	IF NOT (WB_PUD.SF_Close AND WB_PUD.State = 0) THEN WB_PUD.B_Close := TRUE; Init := FALSE; END_IF
	IF NOT (WB_PAF.SF_Close AND WB_PAF.State = 0) THEN WB_PAF.B_Close := TRUE; Init := FALSE; END_IF
	IF NOT (WB_SUD.SF_Close AND WB_SUD.State = 0) THEN WB_SUD.B_Close := TRUE; Init := FALSE; END_IF
	IF NOT (WB_SAF.SF_Close AND WB_SAF.State = 0) THEN WB_SAF.B_Close := TRUE; Init := FALSE; END_IF

	WB_A.B_Close := FALSE;
	WB_B.B_Close := FALSE;
	WB_C.B_Close := FALSE;
	WB_D.B_Close := FALSE;
	WB_E.B_Close := FALSE;
	WB_F.B_Close := FALSE;
	WB_G.B_Close := FALSE;
	WB_H.B_Close := FALSE;
	WB_I.B_Close := FALSE;
	WB_J.B_Close := FALSE;
	WB_K.B_Close := FALSE;
	WB_L.B_Close := FALSE;
	WB_M.B_Close := FALSE;
	WB_N.B_Close := FALSE;
	WB_R.B_Close := FALSE;
	WB_S.B_Close := FALSE;

	WB_PUD.B_Close := FALSE;
	WB_PAF.B_Close := FALSE;
	WB_SUD.B_Close := FALSE;
	WB_SAF.B_Close := FALSE;

	IF NOT (WB_A.SF_Open AND WB_A.State = 0) THEN WB_A.B_Open := TRUE; Init := FALSE; END_IF
	IF NOT (WB_B.SF_Open AND WB_B.State = 0) THEN WB_B.B_Open := TRUE; Init := FALSE; END_IF
	IF NOT (WB_C.SF_Open AND WB_C.State = 0) THEN WB_C.B_Open := TRUE; Init := FALSE; END_IF
	IF NOT (WB_D.SF_Open AND WB_D.State = 0) THEN WB_D.B_Open := TRUE; Init := FALSE; END_IF
	IF NOT (WB_E.SF_Open AND WB_E.State = 0) THEN WB_E.B_Open := TRUE; Init := FALSE; END_IF
	IF NOT (WB_F.SF_Open AND WB_F.State = 0) THEN WB_F.B_Open := TRUE; Init := FALSE; END_IF
	IF NOT (WB_G.SF_Open AND WB_G.State = 0) THEN WB_G.B_Open := TRUE; Init := FALSE; END_IF
	IF NOT (WB_H.SF_Open AND WB_H.State = 0) THEN WB_H.B_Open := TRUE; Init := FALSE; END_IF
	IF NOT (WB_I.SF_Open AND WB_I.State = 0) THEN WB_I.B_Open := TRUE; Init := FALSE; END_IF
	IF NOT (WB_J.SF_Open AND WB_J.State = 0) THEN WB_J.B_Open := TRUE; Init := FALSE; END_IF
	IF NOT (WB_K.SF_Open AND WB_K.State = 0) THEN WB_K.B_Open := TRUE; Init := FALSE; END_IF
	IF NOT (WB_L.SF_Open AND WB_L.State = 0) THEN WB_L.B_Open := TRUE; Init := FALSE; END_IF
	IF NOT (WB_M.SF_Open AND WB_M.State = 0) THEN WB_M.B_Open := TRUE; Init := FALSE; END_IF
	IF NOT (WB_N.SF_Open AND WB_N.State = 0) THEN WB_N.B_Open := TRUE; Init := FALSE; END_IF
	IF NOT (WB_R.SF_Open AND WB_R.State = 0) THEN WB_R.B_Open := TRUE; Init := FALSE; END_IF
	IF NOT (WB_S.SF_Open AND WB_S.State = 0) THEN WB_S.B_Open := TRUE; Init := FALSE; END_IF

	IF NOT (WB_PUD.SF_Open AND WB_PUD.State = 0) THEN WB_PUD.B_Open := TRUE; Init := FALSE; END_IF
	IF NOT (WB_PAF.SF_Open AND WB_PAF.State = 0) THEN WB_PAF.B_Open := TRUE; Init := FALSE; END_IF
	IF NOT (WB_SUD.SF_Open AND WB_SUD.State = 0) THEN WB_SUD.B_Open := TRUE; Init := FALSE; END_IF
	IF NOT (WB_SAF.SF_Open AND WB_SAF.State = 0) THEN WB_SAF.B_Open := TRUE; Init := FALSE; END_IF

*)
END_FUNCTION_BLOCK

(* POU FB/FB_WB_VALVE, ST *)
FUNCTION_BLOCK FB_WB_VALVE
VAR_INPUT
	Enable : BOOL;
	Manual : BOOL;

	B_Open  : BOOL;
	B_Close : BOOL;
	SF_Open  : BOOL;
	SF_Close : BOOL;

END_VAR
VAR_IN_OUT
	P   : ST_SENSOR_BAR;
	CFG : ST_WB_VALVE_CFG;
END_VAR
VAR_OUTPUT
	OUT_Open  : BOOL;
	OUT_Close : BOOL;

	OUT_HP    : BYTE;
END_VAR
VAR
	State : WORD;

	IN_Hmi_Open  : BOOL;
	IN_Hmi_Close : BOOL;

	SI_Open  : FB_SMART_INPUT;
	SI_Close : FB_SMART_INPUT;

	SI_Hmi_Open  : FB_SMART_INPUT;
	SI_Hmi_Close : FB_SMART_INPUT;

	TimeCnt : REAL;
	TimeOut : BOOL;

END_VAR
(*Check Inputs*)
SI_Open (In:= B_Open , T_Cont:= T#0ms, T_DClk:= T#0ms);
SI_Close(In:= B_Close, T_Cont:= T#0ms, T_DClk:= T#0ms);

SI_Hmi_Open (In:= IN_Hmi_Open , T_Cont:= T#0ms, T_DClk:= T#0ms);
SI_Hmi_Close(In:= IN_Hmi_Close, T_Cont:= T#0ms, T_DClk:= T#0ms);

IF NOT Enable THEN
	OUT_Open  := FALSE;
	OUT_Close := FALSE;
	OUT_HP    := 0;

	TimeCnt := 0.0;
	State   := 0;
	RETURN;
END_IF

(*Check Time*)
TimeOut := TimeOut OR ( CFG.TimeMax > 0  AND TimeCnt > CFG.TimeMax );
TimeCnt := TimeCnt + CFG.Cycle;

(*Working States*)
CASE State OF

(*Init State*)
0:
	OUT_Open  := FALSE;
	OUT_Close := FALSE;
	OUT_HP    := 0;

	(*Manual*)
	IF Manual THEN
		IF SI_Hmi_Open.Event = INIT_CONTINUOUS AND NOT P.AlMax THEN
			OUT_Open  := TRUE;
			OUT_HP    := 1;
	
			TimeOut := FALSE; (*Reset TimeOut Error*)
			State   := 1001;  (*Next State*)

		ELSIF SI_Hmi_Close.Event = INIT_CONTINUOUS AND NOT P.AlMax THEN
			OUT_Close := TRUE;
			OUT_HP    := 1;

			TimeOut := FALSE; (*Reset TimeOut Error*)
			State   := 1002;  (*Next State*)

		END_IF

	(*Automatico*)
	ELSE
		IF SI_Open.Event = INIT_CONTINUOUS AND NOT P.AlMax THEN
			OUT_Open  := TRUE;
			OUT_HP    := CFG.HP;

			TimeOut := FALSE; (*Reset TimeOut Error*)
			State   := 1010;  (*Next State*)

		ELSIF SI_Close.Event = INIT_CONTINUOUS AND NOT P.AlMax THEN
			OUT_Close := TRUE;
			OUT_HP    := CFG.HP;

			TimeOut := FALSE; (*Reset TimeOut Error*)
			State   := 1020;  (*Next State*)

		END_IF
	END_IF

    TimeCnt := 0.0; (*Time Count*)

(*Manual OPEN*)
1001:
	(*End*)
	IF SI_Hmi_Open.Event <> NONE OR SI_Hmi_Close.Event <> NONE OR TimeOut OR NOT Manual OR P.AlMax THEN
		OUT_Open  := FALSE;
		OUT_HP    := 0;
		State     := 0; (*Next State*)

	END_IF

(*Manual CLOSE*)
1002:
	(*End*)
	IF SI_Hmi_Open.Event <> NONE OR SI_Hmi_Close.Event <> NONE OR TimeOut OR NOT Manual OR P.AlMax THEN
		OUT_Close := FALSE;
		OUT_HP    := 0;
		State     := 0; (*Next State*)

	END_IF

(*Auto OPEN*)
1010:
	(*End*)
	IF SI_Open.Event <> NONE OR TimeOut OR Manual OR P.AlMax THEN
		OUT_Open  := FALSE;
		OUT_HP    := 0;
		State     := 0; (*Next State*)

	ELSIF SI_Close.Event = INIT_CONTINUOUS THEN
		OUT_Open  := FALSE;
		OUT_Close := TRUE;
		State     := 1020; (*Next State*)

	ELSIF SF_Open THEN
		TimeCnt   := 0.0;
		State     := 1011; (*Next State*)

	END_IF

(*Push OPEN*)
1011:
	(*End*)
	IF SI_Open.Event <> NONE OR TimeOut OR TimeCnt > CFG.PushTime OR (CFG.PushP > 0 AND P.Bar > CFG.PushP) OR Manual OR P.AlMax THEN
		OUT_Open  := FALSE;
		OUT_HP    := 0;
		State     := 0; (*Next State*)

	ELSIF SI_Close.Event = INIT_CONTINUOUS THEN
		OUT_Open  := FALSE;
		OUT_Close := TRUE;
		State     := 1020; (*Next State*)

	END_IF

(*Auto CLOSE*)
1020:
	(*End*)
	IF SI_Close.Event <> NONE OR TimeOut OR Manual OR P.AlMax THEN
		OUT_Close := FALSE;
		OUT_HP    := 0;
		State     := 0; (*Next State*)

	ELSIF SI_Open.Event = INIT_CONTINUOUS THEN
		OUT_Close := FALSE;
		OUT_Open  := TRUE;
		State     := 1010; (*Next State*)

	ELSIF SF_Close THEN
		TimeCnt   := 0.0;
		State     := 1021; (*Next State*)

	END_IF

(*Push CLOSE*)
1021:
	(*End*)
	IF SI_Close.Event <> NONE OR TimeOut OR TimeCnt > CFG.PushTime OR (CFG.PushP > 0 AND P.Bar > CFG.PushP) OR Manual OR P.AlMax THEN
		OUT_Close := FALSE;
		OUT_HP    := 0;
		State     := 0; (*Next State*)

	ELSIF SI_Open.Event = INIT_CONTINUOUS THEN
		OUT_Close := FALSE;
		OUT_Open  := TRUE;
		State     := 1010; (*Next State*)

	END_IF


END_CASE
END_FUNCTION_BLOCK

(* POU FB/FB_WB_VALVE_LS, ST *)
FUNCTION_BLOCK FB_WB_VALVE_LS
VAR_INPUT
	Enable : BOOL;
	Manual : BOOL;

	B_Open  : BOOL;
	B_Half  : BOOL;
	B_Close : BOOL;

	R_Open  : BOOL;
	R_Close : BOOL;

END_VAR
VAR_IN_OUT
	P   : ST_SENSOR_BAR;
	LS  : ST_SENSOR_POS;
	CFG : ST_WB_VALVE_LS_CFG;
END_VAR
VAR_OUTPUT
	OUT_Open  : BOOL;
	OUT_Close : BOOL;

	OUT_HP    : BYTE;
END_VAR
VAR
	State : WORD;

	IN_Hmi_Open  : BOOL;
	IN_Hmi_Close : BOOL;

	SI_Open  : FB_SMART_INPUT;
	SI_Half  : FB_SMART_INPUT;
	SI_Close : FB_SMART_INPUT;

	SI_Hmi_Open  : FB_SMART_INPUT;
	SI_Hmi_Close : FB_SMART_INPUT;
	SI_HmiR_Open  : FB_SMART_INPUT;
	SI_HmiR_Close : FB_SMART_INPUT;

	TimeCnt : REAL;
	TimeOut : BOOL;

	SF_Open : BOOL;
	SF_Half : BOOL;
	SF_Close : BOOL;

END_VAR
(*Check Inputs*)
SI_Open (In:= B_Open , T_Cont:= T#0ms, T_DClk:= T#0ms);
SI_Half (In:= B_Half , T_Cont:= T#0ms, T_DClk:= T#0ms);
SI_Close(In:= B_Close, T_Cont:= T#0ms, T_DClk:= T#0ms);

SI_Hmi_Open  (In:= IN_Hmi_Open , T_Cont:= T#0ms, T_DClk:= T#0ms);
SI_Hmi_Close (In:= IN_Hmi_Close, T_Cont:= T#0ms, T_DClk:= T#0ms);
SI_HmiR_Open (In:= R_Open , T_Cont:= T#0ms, T_DClk:= T#0ms);
SI_HmiR_Close(In:= R_Close, T_Cont:= T#0ms, T_DClk:= T#0ms);

SF_Open  := NOT LS.Err AND LS.Pos > 100.0 - CFG.LS_DB; 	(*OPEN  -> 100%*)
SF_Half  := NOT LS.Err AND LS.Pos > CFG.TgtLS_Half - CFG.LS_DB; (* CFG.LS_DB > ABS(CFG.TgtLS_Half - LS.Pos);*)
SF_Close := NOT LS.Err AND LS.Pos < CFG.LS_DB;  		(*CLOSE ->   0%*)

IF NOT Enable THEN
	OUT_Open  := FALSE;
	OUT_Close := FALSE;
	OUT_HP    := 0;

	TimeCnt := 0.0;
	State   := 0;
	RETURN;
END_IF

(*Check Time*)
TimeOut := TimeOut OR ( CFG.TimeMax > 0  AND TimeCnt > CFG.TimeMax );
TimeCnt := TimeCnt + CFG.Cycle;

(*Working States*)
CASE State OF

(*Init State*)
0:
	OUT_Open  := FALSE;
	OUT_Close := FALSE;
	OUT_HP    := 0;

	(*Manual*)
	IF Manual AND NOT P.AlMax THEN
		IF SI_Hmi_Open.Event = INIT_CONTINUOUS OR SI_HmiR_Open.Event = INIT_CONTINUOUS THEN
			OUT_Open  := TRUE;
			OUT_HP    := 1;
	
			TimeOut := FALSE; (*Reset TimeOut Error*)
			State   := 1001;  (*Next State*)

		ELSIF SI_Hmi_Close.Event = INIT_CONTINUOUS OR SI_HmiR_Close.Event = INIT_CONTINUOUS THEN
			OUT_Close := TRUE;
			OUT_HP    := 1;

			TimeOut := FALSE; (*Reset TimeOut Error*)
			State   := 1002;  (*Next State*)

		END_IF

	(*Automatico*)
	ELSIF NOT P.AlMax AND NOT LS.Err THEN
		IF SI_Open.Event = INIT_CONTINUOUS THEN
			OUT_Open  := TRUE;
			OUT_HP    := CFG.HP;

			TimeOut := FALSE; (*Reset TimeOut Error*)
			State   := 1010;  (*Next State*)

		ELSIF SI_Close.Event = INIT_CONTINUOUS THEN
			OUT_Close := TRUE;
			OUT_HP    := CFG.HP;

			TimeOut := FALSE; (*Reset TimeOut Error*)
			State   := 1020;  (*Next State*)

		ELSIF SI_Half.Event = INIT_CONTINUOUS THEN
			IF LS.Pos < CFG.TgtLS_Half - CFG.LS_DB THEN
				OUT_Open  := TRUE;
				OUT_HP    := CFG.HP;

				TimeOut := FALSE; (*Reset TimeOut Error*)
				State   := 1030;  (*Next State*)

			ELSIF LS.Pos > CFG.TgtLS_Half + CFG.LS_DB THEN
				OUT_Close := TRUE;
				OUT_HP    := CFG.HP;

				TimeOut := FALSE; (*Reset TimeOut Error*)
				State   := 1040;  (*Next State*)

			END_IF
		END_IF
	END_IF

    TimeCnt := 0.0; (*Time Count*)

(*Manual OPEN*)
1001:
	(*End*)
	IF SI_Hmi_Open.Event <> NONE OR SI_HmiR_Open.Event <> NONE
	OR SI_Hmi_Close.Event <> NONE OR SI_HmiR_Close.Event <> NONE
	OR TimeOut OR NOT Manual OR P.AlMax THEN
		OUT_Open  := FALSE;
		OUT_HP    := 0;
		State     := 0; (*Next State*)

	END_IF

(*Manual CLOSE*)
1002:
	(*End*)
	IF SI_Hmi_Open.Event <> NONE OR SI_HmiR_Open.Event <> NONE
	OR SI_Hmi_Close.Event <> NONE OR SI_HmiR_Close.Event <> NONE
	OR TimeOut OR NOT Manual OR P.AlMax THEN
		OUT_Close := FALSE;
		OUT_HP    := 0;
		State     := 0; (*Next State*)

	END_IF

(*Auto OPEN*)
1010,1030:
	(*End*)
	IF SI_Open.Event <> NONE OR SI_Half.Event <> NONE OR TimeOut OR Manual OR P.AlMax OR LS.Err THEN
		OUT_Open  := FALSE;
		OUT_HP    := 0;
		State     := 0; (*Next State*)

	ELSIF SI_Close.Event = INIT_CONTINUOUS THEN
		OUT_Open  := FALSE;
		OUT_Close := TRUE;
		State     := 1020; (*Next State*)

	ELSIF State = 1030 AND LS.Pos > CFG.TgtLS_Half - CFG.LS_DB THEN
		OUT_Open  := FALSE;
		OUT_HP    := 0;
		State     := 0; (*Next State*)

	ELSIF SF_Open THEN
		TimeCnt   := 0.0;
		State     := 1011; (*Next State*)

	END_IF

(*Push OPEN*)
1011:
	(*End*)
	IF SI_Open.Event <> NONE OR TimeOut OR TimeCnt > CFG.PushTime OR (CFG.PushP > 0 AND P.Bar > CFG.PushP) OR Manual OR P.AlMax THEN
		OUT_Open  := FALSE;
		OUT_HP    := 0;
		State     := 0; (*Next State*)

	ELSIF SI_Close.Event = INIT_CONTINUOUS THEN
		OUT_Open  := FALSE;
		OUT_Close := TRUE;
		State     := 1020; (*Next State*)

	END_IF

(*Auto CLOSE*)
1020,1040:
	(*End*)
	IF SI_Close.Event <> NONE OR SI_Half.Event <> NONE OR TimeOut OR Manual OR P.AlMax OR LS.Err THEN
		OUT_Close := FALSE;
		OUT_HP    := 0;
		State     := 0; (*Next State*)

	ELSIF SI_Open.Event = INIT_CONTINUOUS THEN
		OUT_Close := FALSE;
		OUT_Open  := TRUE;
		State     := 1010; (*Next State*)

	ELSIF State = 1040 AND LS.Pos < CFG.TgtLS_Half + CFG.LS_DB THEN
		OUT_Close := FALSE;
		OUT_HP    := 0;
		State     := 0; (*Next State*)

	ELSIF SF_Close THEN
		TimeCnt   := 0.0;
		State     := 1021; (*Next State*)

	END_IF

(*Push CLOSE*)
1021:
	(*End*)
	IF SI_Close.Event <> NONE OR TimeOut OR TimeCnt > CFG.PushTime OR (CFG.PushP > 0 AND P.Bar > CFG.PushP) OR Manual OR P.AlMax THEN
		OUT_Close := FALSE;
		OUT_HP    := 0;
		State     := 0; (*Next State*)

	ELSIF SI_Open.Event = INIT_CONTINUOUS THEN
		OUT_Close := FALSE;
		OUT_Open  := TRUE;
		State     := 1010; (*Next State*)

	END_IF


END_CASE
END_FUNCTION_BLOCK

(* POU FB/FB_WINCHE_V2, ST *)
FUNCTION_BLOCK FB_WINCHE_V2
VAR_INPUT
	Enable : BOOL;
	Ready  : BOOL;

	Perc : REAL;

	IN_1 : ARRAY[1..4] OF BOOL;
	IN_2 : ARRAY[1..4] OF BOOL;
	IN_3 : BOOL;

	Override : BOOL := FALSE;

END_VAR
VAR_IN_OUT
	P_A : ST_SENSOR_BAR;
	P_B : ST_SENSOR_BAR;
	CFG : ST_WINCHE_CFG;
	RAMP: ST_WINCHE_RAMP_CFG;
END_VAR
VAR_OUTPUT
	OUT_TWC : INT;
	OUT_LP  : BYTE;
END_VAR
VAR
	State : WORD;

	IN_SelA : REAL;
	IN_SelB : REAL;
	IN_MaxA : REAL;
	IN_MaxB : REAL;

	IN_Hmi_1 : BOOL;
	IN_Hmi_2 : BOOL;

	SI_A : ARRAY[1..5] OF FB_SMART_INPUT;
	SI_B : ARRAY[1..5] OF FB_SMART_INPUT;

	EventA : EN_SMART_INPUT_STATE;
	EventB : EN_SMART_INPUT_STATE;

	Spd_Tgt  : REAL;
	SoftStop : BOOL;
	Boost    : BOOL;

	CyclCnt : REAL;
	TimeOut : BOOL;

	IsIN_3     : BOOL;
	IsIN_3_Cnt : REAL;

	SpdA : INT;
	SpdB : INT;
	Spd1 : STRING;
	Spd2 : STRING;
	Out_1: BOOL;
	Out_2: BOOL;

	ToFaroInput  : REAL;
	ToFaroOutput : REAL;
END_VAR
IF IN_3 THEN
	IsIN_3     := TRUE;
	IsIN_3_Cnt := 0;
ELSE
	IF IsIN_3_Cnt > 0.25 THEN
		IsIN_3 := FALSE;
	ELSE
		IsIN_3_Cnt := IsIN_3_Cnt + CFG.Cycle;
	END_IF
END_IF


IF Cfg.A_Spd1 THEN
	SpdA := 1;
	SpdB := 2;
	Spd1 := 'A';
	Spd2 := 'B';

	SI_A[1](In:= IN_1[1], T_Cont:= T#0ms, T_DClk:= T#0ms);
	SI_A[2](In:= IN_1[2], T_Cont:= T#0ms, T_DClk:= T#0ms);
	SI_A[3](In:= IN_1[3], T_Cont:= T#0ms, T_DClk:= T#0ms);
	SI_A[4](In:= IN_1[4], T_Cont:= T#0ms, T_DClk:= T#0ms);
	SI_A[5](In:= IN_Hmi_1, T_Cont:= T#0ms, T_DClk:= T#0ms);


	SI_B[1](In:= IN_2[1], T_Cont:= T#0ms, T_DClk:= T#0ms);
	SI_B[2](In:= IN_2[2], T_Cont:= T#0ms, T_DClk:= T#0ms);
	SI_B[3](In:= IN_2[3], T_Cont:= T#0ms, T_DClk:= T#0ms);
	SI_B[4](In:= IN_2[4], T_Cont:= T#0ms, T_DClk:= T#0ms);
	SI_B[5](In:= IN_Hmi_2, T_Cont:= T#0ms, T_DClk:= T#0ms);

	IF    SI_A[1].Event <> NONE THEN EventA := SI_A[1].Event;
	ELSIF SI_A[2].Event <> NONE THEN EventA := SI_A[2].Event;
	ELSIF SI_A[3].Event <> NONE THEN EventA := SI_A[3].Event;
	ELSIF SI_A[4].Event <> NONE THEN EventA := SI_A[4].Event;
	ELSIF SI_A[5].Event <> NONE THEN EventA := SI_A[5].Event;
	ELSE							 EventA := NONE;
	END_IF

	IF    SI_B[1].Event <> NONE THEN EventB := SI_B[1].Event;
	ELSIF SI_B[2].Event <> NONE THEN EventB := SI_B[2].Event;
	ELSIF SI_B[3].Event <> NONE THEN EventB := SI_B[3].Event;
	ELSIF SI_B[4].Event <> NONE THEN EventB := SI_B[4].Event;
	ELSIF SI_B[5].Event <> NONE THEN EventB := SI_B[5].Event;
	ELSE							 EventB := NONE;
	END_IF

	IF IsIN_3 THEN
		IN_SelA := CFG.Spd3[1];
		IN_MaxA := CFG.Spd3[7];

		P_A.MaxBar := CFG.P3_Max;
	ELSE
		IN_SelA := CFG.Spd1[1];
		IN_MaxA := CFG.Spd1[7];

		P_A.MaxBar := CFG.P1_Max;
	END_IF

	IN_SelB := CFG.Spd2[1];
	IN_MaxB := CFG.Spd2[7];

	P_B.MaxBar := CFG.P2_Max;

ELSE
	SpdA := 2;
	SpdB := 1;
	Spd1 := 'B';
	Spd2 := 'A';

	SI_A[1](In:= IN_2[1], T_Cont:= T#0ms, T_DClk:= T#0ms);
	SI_A[2](In:= IN_2[2], T_Cont:= T#0ms, T_DClk:= T#0ms);
	SI_A[3](In:= IN_2[3], T_Cont:= T#0ms, T_DClk:= T#0ms);
	SI_A[4](In:= IN_2[4], T_Cont:= T#0ms, T_DClk:= T#0ms);
	SI_A[5](In:= IN_Hmi_2, T_Cont:= T#0ms, T_DClk:= T#0ms);

	SI_B[1](In:= IN_1[1], T_Cont:= T#0ms, T_DClk:= T#0ms);
	SI_B[2](In:= IN_1[2], T_Cont:= T#0ms, T_DClk:= T#0ms);
	SI_B[3](In:= IN_1[3], T_Cont:= T#0ms, T_DClk:= T#0ms);
	SI_B[4](In:= IN_1[4], T_Cont:= T#0ms, T_DClk:= T#0ms);
	SI_B[5](In:= IN_Hmi_1, T_Cont:= T#0ms, T_DClk:= T#0ms);

	IF    SI_A[1].Event <> NONE THEN EventA := SI_A[1].Event;
	ELSIF SI_A[2].Event <> NONE THEN EventA := SI_A[2].Event;
	ELSIF SI_A[3].Event <> NONE THEN EventA := SI_A[3].Event;
	ELSIF SI_A[4].Event <> NONE THEN EventA := SI_A[4].Event;
	ELSIF SI_A[5].Event <> NONE THEN EventA := SI_A[5].Event;
	ELSE							 EventA := NONE;
	END_IF

	IF    SI_B[1].Event <> NONE THEN EventB := SI_B[1].Event;
	ELSIF SI_B[2].Event <> NONE THEN EventB := SI_B[2].Event;
	ELSIF SI_B[3].Event <> NONE THEN EventB := SI_B[3].Event;
	ELSIF SI_B[4].Event <> NONE THEN EventB := SI_B[4].Event;
	ELSIF SI_B[5].Event <> NONE THEN EventB := SI_B[5].Event;
	ELSE							 EventB := NONE;
	END_IF

	IF IsIN_3 THEN
		IN_SelB := CFG.Spd3[1];
		IN_MaxB := CFG.Spd3[7];

		P_B.MaxBar := CFG.P3_Max;
	ELSE
		IN_SelB := CFG.Spd1[1];
		IN_MaxB := CFG.Spd1[7];

		P_B.MaxBar := CFG.P1_Max;
	END_IF

	IN_SelA := CFG.Spd2[1];
	IN_MaxA := CFG.Spd2[7];

	P_A.MaxBar := CFG.P2_Max;

END_IF
(*
IF    IN_SpdA < 1 THEN IN_SpdA := 1;
ELSIF IN_SpdA > 7 THEN IN_SpdA := 7;
END_IF

IF    IN_SpdB < 1 THEN IN_SpdB := 1;
ELSIF IN_SpdB > 7 THEN IN_SpdB := 7;
END_IF
*)
ToFaroInput := 0.0;
IF IN_1[1] OR IN_1[2] OR IN_1[3] OR IN_1[4] OR IN_Hmi_1 THEN ToFaroInput := 1.0;               END_IF
IF IN_2[1] OR IN_2[2] OR IN_2[3] OR IN_2[4] OR IN_Hmi_2 THEN ToFaroInput := 2.0 + ToFaroInput; END_IF

IF NOT Enable THEN
	OUT_TWC := 0;
	OUT_LP  := 0;

	CyclCnt := 0;
	State   := 0;
	RETURN;
END_IF

(*Check Time*)
TimeOut := TimeOut OR (CFG.TimeMax > 0 AND CyclCnt > CFG.TimeMax);
CyclCnt := CyclCnt + CFG.Cycle;

CASE State OF
0: (*INIT*)
	OUT_TWC := 0;
	CyclCnt := 0;

	SoftStop := FALSE;
	Boost    := FALSE;

	IF Ready THEN
		IF EventA = INIT_CONTINUOUS AND NOT P_A.AlMax THEN
			Spd_Tgt := RAMP.Spd_Min;
			OUT_TWC := REAL_TO_INT(Spd_Tgt * Perc * 10.0);
			TimeOut := FALSE;
			State   := 10;

		ELSIF EventB = INIT_CONTINUOUS AND NOT P_B.AlMax THEN
			Spd_Tgt := RAMP.Spd_Min;
			OUT_TWC := REAL_TO_INT(-Spd_Tgt * Perc * 10.0);
			TimeOut := FALSE;
			State   := 20;

		END_IF
	END_IF


10: (*A*)
	IF TimeOut OR P_A.AlMax THEN
		OUT_TWC := 0;
		State   := 0;

	ELSE
		IF EventA = INIT_CONTINUOUS THEN
			SoftStop := FALSE;
			CyclCnt  := 0;
		ELSIF EventA = END_CONTINUOUS THEN
			SoftStop := TRUE;
		END_IF

		IF SoftStop THEN
			IF EventB = INIT_CONTINUOUS THEN
				Spd_Tgt := RAMP.Spd_Min;
				OUT_TWC := REAL_TO_INT(-Spd_Tgt * Perc * 10.0);
				TimeOut := FALSE;
				State   := 20;

			ELSE
				Spd_Tgt := Spd_Tgt - RAMP.Spd_Dec * CFG.Cycle;
				Spd_Tgt := MIN(Spd_Tgt, IN_SelA     );
				Spd_Tgt := MAX(Spd_Tgt, RAMP.Spd_Min);

				IF Spd_Tgt = RAMP.Spd_Min OR RAMP.Spd_Dec <= 0
				THEN OUT_TWC := 0;
				ELSE OUT_TWC := REAL_TO_INT(Spd_Tgt * Perc * 10.0);
				END_IF

			END_IF

		ELSE
			IF EventB = INIT_CONTINUOUS OR Override THEN
				Boost := TRUE;
			ELSIF EventB = END_CONTINUOUS THEN
				Boost := FALSE;
			END_IF

			Spd_Tgt := Spd_Tgt + RAMP.Spd_Inc * CFG.Cycle;
			IF Boost
			THEN Spd_Tgt := MIN(Spd_Tgt, IN_MaxA );
			ELSE Spd_Tgt := MIN(Spd_Tgt, IN_SelA );
			END_IF
			Spd_Tgt := MAX(Spd_Tgt, RAMP.Spd_Min);

			OUT_TWC := REAL_TO_INT(Spd_Tgt * Perc * 10.0);

		END_IF

		IF OUT_TWC = 0 THEN
			State    := 0; (*Next State*)
		END_IF

		(*OUT_TWC := REAL_TO_INT(CFG.SpdA[IN_SpdA] * Perc * 10.0);*)

	END_IF

20: (*B*)
	IF TimeOut OR P_B.AlMax THEN
		OUT_TWC := 0;
		State   := 0;

	ELSE
		IF EventB = INIT_CONTINUOUS THEN
			SoftStop := FALSE;
			CyclCnt  := 0;
		ELSIF EventB = END_CONTINUOUS THEN
			SoftStop := TRUE;
		END_IF

		IF SoftStop THEN
			IF EventA = INIT_CONTINUOUS THEN
				Spd_Tgt := RAMP.Spd_Min;
				OUT_TWC := REAL_TO_INT(Spd_Tgt * Perc * 10.0);
				TimeOut := FALSE;
				State   := 10;

			ELSE
				Spd_Tgt := Spd_Tgt - RAMP.Spd_Dec * CFG.Cycle;
				Spd_Tgt := MIN(Spd_Tgt, IN_SelB     );
				Spd_Tgt := MAX(Spd_Tgt, RAMP.Spd_Min);
	
				IF Spd_Tgt = RAMP.Spd_Min OR RAMP.Spd_Dec <= 0
				THEN OUT_TWC := 0;
				ELSE OUT_TWC := REAL_TO_INT(-Spd_Tgt * Perc * 10.0);
				END_IF

			END_IF

		ELSE
			IF EventA = INIT_CONTINUOUS OR Override THEN
				Boost := TRUE;
			ELSIF EventA = END_CONTINUOUS THEN
				Boost := FALSE;
			END_IF

			Spd_Tgt := Spd_Tgt + RAMP.Spd_Inc * CFG.Cycle;
			IF Boost
			THEN Spd_Tgt := MIN(Spd_Tgt, IN_MaxB );
			ELSE Spd_Tgt := MIN(Spd_Tgt, IN_SelB );
			END_IF
			Spd_Tgt := MAX(Spd_Tgt, RAMP.Spd_Min);

			OUT_TWC := REAL_TO_INT(-Spd_Tgt * Perc * 10.0);

		END_IF

		IF OUT_TWC = 0 THEN
			State    := 0; (*Next State*)
		END_IF

		(*OUT_TWC := REAL_TO_INT(-CFG.SpdB[IN_SpdB] * Perc * 10.0);*)

	END_IF

END_CASE

IF Cfg.A_Spd1 THEN
	Out_1 := OUT_TWC > 0;
	Out_2 := OUT_TWC < 0;
ELSE
	Out_1 := OUT_TWC < 0;
	Out_2 := OUT_TWC > 0;
END_IF

IF OUT_TWC = 0 THEN
	OUT_LP := 0;
ELSE
	OUT_LP  := 1; (*How Many*)
END_IF

(*Gear to FARO*)
IF Out_1 THEN
	IF IsIN_3
	THEN ToFaroOutput := 1;
	ELSE ToFaroOutput := 3;
	END_IF
ELSIF Out_2 THEN
	ToFaroOutput := 2;
ELSE
	ToFaroOutput := 0;
END_IF
END_FUNCTION_BLOCK

(* POU FB/FB_BOARD, ST *)
FUNCTION_BLOCK FB_BOARD
VAR_INPUT
	Enable : BOOL;
	Ready  : BOOL;

	EngReady : BOOL;
	Latching : BOOL;

	Keel_Pos : REAL;
	Keel_Err : BOOL;

	IN_P : ARRAY[1..2] OF BOOL;
	IN_S : ARRAY[1..2] OF BOOL;
	IN_C : ARRAY[1..2] OF BOOL;

END_VAR
VAR_IN_OUT
	PA_P : ST_SENSOR_BAR;
	PA_S : ST_SENSOR_BAR;
	PB_P : ST_SENSOR_BAR;
	PB_S : ST_SENSOR_BAR;

	LS_P : ST_SENSOR_POS;
	LS_S : ST_SENSOR_POS;

	SF_P : ST_SENSOR_SWITCH;
	SF_S : ST_SENSOR_SWITCH;

	CFG : ST_BOARD_CFG;
END_VAR
VAR_OUTPUT
	OUT_TWC_P : INT;
	OUT_TWC_S : INT;

	OUT_EVB_P : BOOL;
	OUT_EVB_S : BOOL;

	OUT_EVT_P : BOOL;
	OUT_EVT_S : BOOL;

	OUT_LP : BYTE;

END_VAR
VAR
	State   : WORD;

	IN_Hmi_P : BOOL;
	IN_Hmi_S : BOOL;
	IN_Hmi_C : BOOL;

	IN_Hmi_P_In  : BOOL;
	IN_Hmi_S_In  : BOOL;
	IN_Hmi_P_Out : BOOL;
	IN_Hmi_S_Out : BOOL;

	IN_Hmi_InPerc  : INT := 20;
	IN_Hmi_OutPerc : INT := 20;

	SI_P : ARRAY[1..3] OF FB_SMART_INPUT;
	SI_S : ARRAY[1..3] OF FB_SMART_INPUT;
	SI_C : ARRAY[1..3] OF FB_SMART_INPUT;

	Event_P : EN_SMART_INPUT_STATE;
	Event_S : EN_SMART_INPUT_STATE;
	Event_C : EN_SMART_INPUT_STATE;

	SI_P_In  : FB_SMART_INPUT;
	SI_S_In  : FB_SMART_INPUT;
	SI_P_Out : FB_SMART_INPUT;
	SI_S_Out : FB_SMART_INPUT;

	TimeCnt : REAL;
	TimeOut : BOOL;

	P_Alarm: BOOL;

	TWC_P_Inc : REAL;
	TWC_S_Inc : REAL;


	LS_Err : BOOL;

	P_Bypass  : BOOL;

	Slow : BOOL;
	LS_Dif : REAL;

	LS_P_Out : BOOL;
	LS_S_Out : BOOL;
	LS_P_In  : BOOL;
	LS_S_In  : BOOL;
	LS_P_Mid : BOOL;
	LS_S_Mid : BOOL;

	LS_Safe_P_Out : BOOL;
	LS_Safe_S_Out : BOOL;
	LS_Safe_P_In  : BOOL;
	LS_Safe_S_In  : BOOL;


	MOVING_P : BOOL;
	MOVING_C : BOOL;
	MOVING_S : BOOL;

	MOVING_P_In  : BOOL;
	MOVING_P_Out : BOOL;
	MOVING_S_In  : BOOL;
	MOVING_S_Out : BOOL;

	Out_IN  : BOOL;
(*	Out_IN1 : BOOL;
	Out_IN2 : BOOL;
	Out_IN3 : BOOL;*)
	Out_OUT : BOOL;


	DeltaP  : REAL;
	DeltaS  : REAL;
	DeltaPS : REAL;

	SoftStop: BOOL;

	Hyst_Cnt : REAL;
	Hyst_ON  : BOOL;

END_VAR
VAR PERSISTENT
	Manual AT %Q*: BOOL;

	Hatch_Enable AT %Q*: BOOL;
END_VAR
P_Alarm := PA_P.AlMax OR PA_S.AlMax OR PB_P.AlMax OR PB_S.AlMax;
LS_Err  := LS_P.Err OR LS_S.Err;

LS_P_In  := NOT LS_P.Err AND LS_P.Pos > CFG.TgtLS_P_In  - CFG.LS_DB;
LS_P_Out := NOT LS_P.Err AND LS_P.Pos < CFG.TgtLS_P_Out + CFG.LS_DB;
LS_P_Mid := NOT LS_P.Err AND LS_P.Pos > CFG.TgtLS_P_Mid - CFG.LS_DB AND LS_P.Pos < CFG.TgtLS_P_Mid + CFG.LS_DB;

LS_S_In  := NOT LS_S.Err AND LS_S.Pos > CFG.TgtLS_S_In  - CFG.LS_DB;
LS_S_Out := NOT LS_S.Err AND LS_S.Pos < CFG.TgtLS_S_Out + CFG.LS_DB;
LS_S_Mid := NOT LS_S.Err AND LS_S.Pos > CFG.TgtLS_S_Mid - CFG.LS_DB AND LS_S.Pos < CFG.TgtLS_S_Mid + CFG.LS_DB;

LS_Safe_P_In  := NOT LS_P.Err AND LS_P.Pos > CFG.TgtLS_P_Safe_In  - CFG.LS_DB;
LS_Safe_P_Out := NOT LS_P.Err AND LS_P.Pos < CFG.TgtLS_P_Safe_Out + CFG.LS_DB;

LS_Safe_S_In  := NOT LS_S.Err AND LS_S.Pos > CFG.TgtLS_S_Safe_In  - CFG.LS_DB;
LS_Safe_S_Out := NOT LS_S.Err AND LS_S.Pos < CFG.TgtLS_S_Safe_Out + CFG.LS_DB;

SI_P[1](In:= IN_P[1],  T_Cont:= T#0ms, T_DClk:= T#0ms);
SI_P[2](In:= IN_P[2],  T_Cont:= T#0ms, T_DClk:= T#0ms);
SI_P[3](In:= IN_Hmi_P, T_Cont:= T#0ms, T_DClk:= T#0ms);

SI_S[1](In:= IN_S[1],  T_Cont:= T#0ms, T_DClk:= T#0ms);
SI_S[2](In:= IN_S[2],  T_Cont:= T#0ms, T_DClk:= T#0ms);
SI_S[3](In:= IN_Hmi_S, T_Cont:= T#0ms, T_DClk:= T#0ms);

SI_C[1](In:= IN_C[1],  T_Cont:= T#0ms, T_DClk:= T#0ms);
SI_C[2](In:= IN_C[2],  T_Cont:= T#0ms, T_DClk:= T#0ms);
SI_C[3](In:= IN_Hmi_C, T_Cont:= T#0ms, T_DClk:= T#0ms);

SI_P_In (In:= IN_Hmi_P_In,  T_Cont:= T#0ms, T_DClk:= T#0ms);
SI_S_In (In:= IN_Hmi_S_In,  T_Cont:= T#0ms, T_DClk:= T#0ms);
SI_P_Out(In:= IN_Hmi_P_Out, T_Cont:= T#0ms, T_DClk:= T#0ms);
SI_S_Out(In:= IN_Hmi_S_Out, T_Cont:= T#0ms, T_DClk:= T#0ms);

IF NOT Enable THEN
	OUT_TWC_P := 0;
	OUT_TWC_S := 0;

	OUT_EVB_P := FALSE;
	OUT_EVB_S := FALSE;

	OUT_EVT_P := FALSE;
	OUT_EVT_S := FALSE;

	OUT_LP := 0;

	MOVING_P := FALSE;
	MOVING_C := FALSE;
	MOVING_S := FALSE;

	MOVING_P_In  := FALSE;
	MOVING_P_Out := FALSE;
	MOVING_S_In  := FALSE;
	MOVING_S_Out := FALSE;

	TimeCnt := 0.0;
	State   := 0;
	RETURN;
END_IF

(*Check Time*)
TimeOut := TimeOut OR ( CFG.TimeMax > 0  AND TimeCnt > CFG.TimeMax );
TimeCnt := TimeCnt + CFG.Cycle;

IF    SI_P[1].Event <> NONE THEN Event_P := SI_P[1].Event;
ELSIF SI_P[2].Event <> NONE THEN Event_P := SI_P[2].Event;
ELSIF SI_P[3].Event <> NONE THEN Event_P := SI_P[3].Event;
ELSE							 Event_P := NONE;
END_IF

IF    SI_S[1].Event <> NONE THEN Event_S := SI_S[1].Event;
ELSIF SI_S[2].Event <> NONE THEN Event_S := SI_S[2].Event;
ELSIF SI_S[3].Event <> NONE THEN Event_S := SI_S[3].Event;
ELSE							 Event_S := NONE;
END_IF

IF    SI_C[1].Event <> NONE THEN Event_C := SI_C[1].Event;
ELSIF SI_C[2].Event <> NONE THEN Event_C := SI_C[2].Event;
ELSIF SI_C[3].Event <> NONE THEN Event_C := SI_C[3].Event;
ELSE							 Event_C := NONE;
END_IF

(*Working States*)
CASE State OF
0:
	OUT_TWC_P := 0;
	OUT_TWC_S := 0;

	OUT_EVB_P := FALSE;
	OUT_EVB_S := FALSE;

	OUT_EVT_P := FALSE;
	OUT_EVT_S := FALSE;

	OUT_LP := 0;

	MOVING_P_In  := FALSE;
	MOVING_P_Out := FALSE;
	MOVING_S_In  := FALSE;
	MOVING_S_Out := FALSE;

	MOVING_P := FALSE;
	MOVING_C := FALSE;
	MOVING_S := FALSE;

	SoftStop := FALSE;
	Hyst_cnt := CFG.P_Hyst_TM + CFG.Cycle;

	IF Manual AND Ready THEN
		(*Manual Port IN -> Cylinder Out*)
		IF SI_P_In.Event = INIT_CONTINUOUS AND NOT SF_P.Alarm.Alarm THEN
			MOVING_P_In := TRUE;
			TWC_P_Inc   := -CFG.EVP_In_P_Min;

			TimeOut := FALSE; (*Reset TimeOut Error*)
			State   := 100;   (*Next State*)

		(*Manual Port OUT -> Cylinder In*)
		ELSIF SI_P_Out.Event = INIT_CONTINUOUS THEN
			MOVING_P_Out := TRUE;
			TWC_P_Inc    := CFG.EVP_Out_P_Min;

			TimeOut  := FALSE; (*Reset TimeOut Error*)
			State    := 200;   (*Next State*)

		(*Manual Stbd IN -> Cylinder Out*)
		ELSIF SI_S_In.Event = INIT_CONTINUOUS AND NOT SF_S.Alarm.Alarm THEN
			MOVING_S_In := TRUE;
			TWC_S_Inc   := -CFG.EVP_In_S_Min;

			TimeOut := FALSE; (*Reset TimeOut Error*)
			State   := 300;   (*Next State*)

		(*Manual Stbd OUT -> Cylinder In*)
		ELSIF SI_S_Out.Event = INIT_CONTINUOUS THEN
			MOVING_S_Out := TRUE;
			TWC_S_Inc    := CFG.EVP_Out_S_Min;

			TimeOut := FALSE; (*Reset TimeOut Error*)
			State   := 400;   (*Next State*)

		END_IF

	ELSIF Ready AND NOT LS_Err THEN

		IF Event_P = INIT_CONTINUOUS THEN

			IF LS_P_Out AND LS_S_In AND NOT SF_P.Alarm.Alarm THEN
				MOVING_S  := TRUE;
				TWC_P_Inc := -CFG.EVP_In_P_Min;  (*Port IN  -> Cylinder Out*)
				TWC_S_Inc :=  CFG.EVP_Out_S_Min; (*Stbd OUT -> Cylinder In*)

				TimeOut := FALSE; (*Reset TimeOut Error*)
				State   := 6000;  (*Retracted Port*)

			ELSIF NOT SF_S.Alarm.Alarm THEN
				MOVING_P  := TRUE;
				TWC_P_Inc :=  CFG.EVP_Out_P_Min; (*Port OUT -> Cylinder In*)
				TWC_S_Inc := -CFG.EVP_In_S_Min;  (*Stbd IN  -> Cylinder Out*)

				TimeOut := FALSE; (*Reset TimeOut Error*)
				State   := 1000;  (*Full Port*)
			END_IF

		ELSIF Event_S = INIT_CONTINUOUS THEN

			IF LS_P_In AND LS_S_Out AND NOT SF_S.Alarm.Alarm THEN
				MOVING_P  := TRUE;
				TWC_P_Inc :=  CFG.EVP_Out_P_Min; (*Port OUT -> Cylinder In*)
				TWC_S_Inc := -CFG.EVP_In_S_Min;  (*Stbd IN  -> Cylinder Out*)

				TimeOut := FALSE; (*Reset TimeOut Error*)
				State   := 5000;  (*Retracted Stbd*)

			ELSIF NOT SF_P.Alarm.Alarm THEN
				MOVING_S  := TRUE;
				TWC_P_Inc := -CFG.EVP_In_P_Min;  (*Port IN  -> Cylinder Out*)
				TWC_S_Inc :=  CFG.EVP_Out_S_Min; (*Stbd OUT -> Cylinder In*)

				TimeOut := FALSE; (*Reset TimeOut Error*)
				State   := 2000;  (*Full Stbd*)

			END_IF

		ELSIF Event_C = INIT_CONTINUOUS THEN
			MOVING_C  := TRUE;

			IF LS_P.Pos > CFG.TgtLS_P_Mid + CFG.LS_DB OR LS_S.Pos < CFG.TgtLS_S_Mid - CFG.LS_DB THEN
				MOVING_P  := TRUE;
				TWC_P_Inc :=  CFG.EVP_Out_P_Min;
				TWC_S_Inc := -CFG.EVP_In_S_Min;

				TimeOut := FALSE; (*Reset TimeOut Error*)
				State   := 3000;  (*Next State*)

			ELSIF LS_P.Pos < CFG.TgtLS_P_Mid - CFG.LS_DB OR LS_S.Pos > CFG.TgtLS_S_Mid + CFG.LS_DB THEN
				MOVING_S  := TRUE;
				TWC_P_Inc := -CFG.EVP_In_P_Min; (*Port IN -> Cylinder Out*)
				TWC_S_Inc :=  CFG.EVP_Out_S_Min;

				TimeOut := FALSE; (*Reset TimeOut Error*)
				State   := 4000;  (*Next State*)

			END_IF
		END_IF
	END_IF

(*Manual Port IN -> Cylinder Out*)
100:
	IF SI_P_In.Event = END_CONTINUOUS OR SI_P_Out.Event = INIT_CONTINUOUS OR NOT Ready OR SF_P.Alarm.Alarm OR TimeOut OR P_Alarm THEN
		OUT_TWC_P := 0;
		OUT_LP    := 0;
		State     := 0;

	ELSE
		TWC_P_Inc := MAX(MAX(TWC_P_Inc - CFG.EVP_In_Inc * CFG.Cycle, -IN_Hmi_InPerc), -CFG.EVP_In_P_Max);
		OUT_TWC_P := REAL_TO_INT(TWC_P_Inc * 10.0);
		OUT_LP    := 1;

	END_IF

(*Manual Port OUT -> Cylinder In*)
200:
	IF SI_P_Out.Event = END_CONTINUOUS OR SI_P_In.Event = INIT_CONTINUOUS OR NOT Ready OR TimeOut OR P_Alarm THEN
		OUT_EVB_P := FALSE;
		OUT_EVT_P := FALSE;
		OUT_TWC_P := 0;
		OUT_LP    := 0;
		State     := 0;

	ELSE
		TWC_P_Inc := MIN(MIN(TWC_P_Inc + CFG.EVP_Out_Inc * CFG.Cycle, IN_Hmi_OutPerc), CFG.EVP_Out_P_Max);
		OUT_EVB_P := TRUE;
		OUT_EVT_P := TRUE;
		OUT_TWC_P := REAL_TO_INT(TWC_P_Inc * 10.0);
		OUT_LP    := 1;

	END_IF

(*Manual Stbd IN -> Cylinder Out*)
300:
	IF SI_S_In.Event = END_CONTINUOUS OR SI_S_Out.Event = INIT_CONTINUOUS OR NOT Ready OR SF_S.Alarm.Alarm OR TimeOut OR P_Alarm THEN
		OUT_TWC_S := 0;
		OUT_LP    := 0;
		State     := 0;

	ELSE
		TWC_S_Inc := MAX(MAX(TWC_S_Inc - CFG.EVP_In_Inc * CFG.Cycle, -IN_Hmi_InPerc), -CFG.EVP_In_S_Max);
		OUT_TWC_S := REAL_TO_INT(TWC_S_Inc * 10.0);
		OUT_LP    := 1;

	END_IF

(*Manual Stbd OUT -> Cylinder In*)
400:
	IF SI_S_Out.Event = END_CONTINUOUS OR SI_S_In.Event = INIT_CONTINUOUS OR NOT Ready OR TimeOut OR P_Alarm THEN
		OUT_EVB_S := FALSE;
		OUT_EVT_S := FALSE;
		OUT_TWC_S := 0;
		OUT_LP    := 0;
		State     := 0;

	ELSE
		TWC_S_Inc := MIN(MIN(TWC_S_Inc + CFG.EVP_Out_Inc * CFG.Cycle, IN_Hmi_OutPerc), CFG.EVP_Out_S_Max);
		OUT_EVB_S := TRUE;
		OUT_EVT_S := TRUE;
		OUT_TWC_S := REAL_TO_INT(TWC_S_Inc * 10.0);
		OUT_LP    := 1;

	END_IF

(*Moving to PORT*)
(*Automatic/Momentary Port OUT -> Cylinder In*)
(*Automatic/Momentary Stbd IN  -> Cylinder Out*)
1000, 3000, 5000:

	IF State = 3000 THEN
		DeltaP  := LS_P.Pos - CFG.TgtLS_P_Mid; 		(*Positive*)
		DeltaS  := LS_S.Pos - CFG.TgtLS_S_Mid; 		(*Negative*)
		DeltaPS := DeltaP + DeltaS + CFG.LS_Dif_Tgt;(*Positive -> Out Late*)

	ELSIF State = 5000 THEN
		DeltaP  := LS_P.Pos - CFG.TgtLS_P_InR;		(*Positive*)
		DeltaS  := LS_S.Pos - CFG.TgtLS_S_OutR; 	(*Negative*)
		DeltaPS := DeltaP + DeltaS + CFG.LS_Dif_Tgt;(*Positive -> Out Late*)

	ELSIF Keel_Err OR Keel_Pos > CFG.Keel_P_Max THEN
		DeltaP  := LS_P.Pos - CFG.TgtLS_P_Safe_Out; (*Positive*)
		DeltaS  := LS_S.Pos - CFG.TgtLS_S_Safe_In; 	(*Negative*)
		DeltaPS := DeltaP + DeltaS + CFG.LS_Dif_Tgt;(*Positive -> Out Late*)

	ELSE
		DeltaP  := LS_P.Pos - CFG.TgtLS_P_Out; 		(*Positive*)
		DeltaS  := LS_S.Pos - CFG.TgtLS_S_In; 		(*Negative*)
		DeltaPS := DeltaP + DeltaS + CFG.LS_Dif_Tgt;(*Positive -> Out Late*)

	END_IF

	IF Manual OR NOT Ready OR SF_S.Alarm.Alarm OR LS_Err OR P_Alarm OR TimeOut THEN
		OUT_EVB_P := FALSE;
		OUT_EVT_P := FALSE;
		OUT_TWC_P := 0;
		OUT_TWC_S := 0;
		OUT_LP    := 0;
		State     := 0;

	ELSIF DeltaP <= 0.0 AND DeltaS >= 0.0 THEN
		OUT_EVB_P := FALSE;
		OUT_EVT_P := FALSE;
		OUT_TWC_P := 0;
		OUT_TWC_S := 0;
		OUT_LP    := 0;
		State     := 0;

	ELSE
		(*Activate SoftStop*)
		IF Event_P = INIT_CONTINUOUS OR Event_S = INIT_CONTINUOUS OR Event_C = INIT_CONTINUOUS
		OR State = 1000 AND ((NOT EngReady OR NOT Latching) AND Event_P = END_CONTINUOUS)
		OR State = 3000 AND ((NOT EngReady OR NOT Latching) AND Event_C = END_CONTINUOUS)
		OR State = 5000 AND ((NOT EngReady OR NOT Latching) AND Event_S = END_CONTINUOUS)
		THEN

			IF SoftStop THEN
				OUT_EVB_P := FALSE;
				OUT_EVT_P := FALSE;
				OUT_TWC_P := 0;
				OUT_TWC_S := 0;
				OUT_LP    := 0;
				State     := 0;
				RETURN;

			ELSE
				SoftStop := TRUE;

			END_IF
		END_IF

		(*Port OUT -> Cylinder In*)
		IF SoftStop OR DeltaPS < -CFG.LS_Dif_Max THEN
			TWC_P_Inc := TWC_P_Inc - CFG.EVP_Out_Dec * CFG.Cycle; 						(*Increment*)
			TWC_P_Inc := MIN(TWC_P_Inc, CFG.EVP_Out_P_Max);								(*Max Value*)
			TWC_P_Inc := MIN(TWC_P_Inc, CFG.EVP_Out_P_Min + DeltaP * CFG.EVP_Out_LS_K); (*Approx K*)
			TWC_P_Inc := MAX(TWC_P_Inc, CFG.EVP_Out_P_Min); 							(*Min Value - Extra check*)

			IF TWC_P_Inc = CFG.EVP_Out_P_Min OR CFG.EVP_Out_Dec <= 0 THEN
				OUT_TWC_P := 0;
				OUT_EVB_P := FALSE;
			ELSE
				OUT_TWC_P := REAL_TO_INT(TWC_P_Inc * 10.0);
				OUT_EVB_P := TRUE;
			END_IF

			OUT_EVT_P := FALSE;

		ELSIF DeltaP > 0.0 (*AND DeltaPS > -CFG.LS_Dif_Max*) THEN
			TWC_P_Inc := TWC_P_Inc + CFG.EVP_Out_Inc * CFG.Cycle; 						(*Increment*)
			TWC_P_Inc := MIN(TWC_P_Inc, CFG.EVP_Out_P_Max);								(*Max Value*)
			TWC_P_Inc := MIN(TWC_P_Inc, CFG.EVP_Out_P_Min + DeltaP * CFG.EVP_Out_LS_K); (*Approx K*)

			IF EngReady																	(*Delta K*)
			THEN TWC_P_Inc := MIN(TWC_P_Inc, CFG.EVP_Out_P_Eng + DeltaPS * CFG.EVP_Out_EVP_K);
			ELSE TWC_P_Inc := MIN(TWC_P_Inc, CFG.EVP_Out_P_PP  + DeltaPS * CFG.EVP_Out_EVP_K);
			END_IF

			TWC_P_Inc := MAX(TWC_P_Inc, CFG.EVP_Out_P_Min); 							(*Min Value - Extra check*)

			OUT_TWC_P := REAL_TO_INT(TWC_P_Inc * 10.0);
			OUT_EVB_P := TRUE;

			IF Hyst_Cnt > CFG.P_Hyst_TM THEN
				Hyst_ON := TRUE;
			ELSE
				Hyst_ON  := FALSE;
				Hyst_Cnt := Hyst_Cnt + CFG.Cycle;
			END_IF
	
			IF PB_P.Bar > CFG.P_Hyst_HP AND Hyst_ON OR PB_P.Err THEN
				OUT_EVT_P := TRUE;
				Hyst_cnt  := 0.0;
			ELSIF PB_P.Bar < CFG.P_Hyst_LP AND Hyst_ON THEN
				OUT_EVT_P := FALSE;
				Hyst_cnt  := 0.0;
			END_IF

		ELSE
			OUT_TWC_P := 0;
			OUT_EVB_P := FALSE;
			OUT_EVT_P := FALSE;
		END_IF

		(*Stbd IN  -> Cylinder Out*)
		IF SoftStop OR DeltaPS > CFG.LS_Dif_Min THEN
			TWC_S_Inc := TWC_S_Inc + CFG.EVP_In_Dec * CFG.Cycle; 						(*Increment*)
			TWC_S_Inc := MAX(TWC_S_Inc, -CFG.EVP_In_S_Max); 							(*Max Value*)
			TWC_S_Inc := MAX(TWC_S_Inc, -CFG.EVP_In_S_Min + DeltaS * CFG.EVP_In_LS_K); 	(*Approx K*)
			TWC_S_Inc := MIN(TWC_S_Inc, -CFG.EVP_In_S_Min); 							(*Min Value - Extra check*)

			IF TWC_S_Inc = -CFG.EVP_In_S_Min OR CFG.EVP_In_Dec <= 0
			THEN OUT_TWC_S := 0;
			ELSE OUT_TWC_S := REAL_TO_INT(TWC_S_Inc * 10.0);
			END_IF

		ELSIF DeltaS < 0.0 (*AND DeltaPS < CFG.LS_Dif_Min*) THEN
			TWC_S_Inc := TWC_S_Inc - CFG.EVP_In_Inc * CFG.Cycle; 						(*Increment*)
			TWC_S_Inc := MAX(TWC_S_Inc, -CFG.EVP_In_S_Max); 							(*Max Value*)
			TWC_S_Inc := MAX(TWC_S_Inc, -CFG.EVP_In_S_Min + DeltaS * CFG.EVP_In_LS_K); 	(*Approx K*)

			IF EngReady																	(*Delta K*)
			THEN TWC_S_Inc := MAX(TWC_S_Inc, -CFG.EVP_In_S_Eng + DeltaPS * CFG.EVP_In_EVP_K);
			ELSE TWC_S_Inc := MAX(TWC_S_Inc, -CFG.EVP_In_S_PP  + DeltaPS * CFG.EVP_In_EVP_K);
			END_IF

			TWC_S_Inc := MIN(TWC_S_Inc, -CFG.EVP_In_S_Min); 							(*Min Value - Extra check*)

			OUT_TWC_S := REAL_TO_INT(TWC_S_Inc * 10.0);

		ELSE
			OUT_TWC_S := 0;

		END_IF

		OUT_LP := CFG.LP;

		(*If both stopped go to Init State*)
		IF OUT_TWC_P = 0 AND OUT_TWC_S = 0 THEN
			OUT_EVB_P := FALSE;
			OUT_EVT_P := FALSE;
			OUT_TWC_P := 0;
			OUT_TWC_S := 0;
			OUT_LP    := 0;
			State     := 0;

		END_IF

	END_IF


(*Moving to STBD*)
(*Automatic/Momentary Port IN  -> Cylinder Out*)
(*Automatic/Momentary Stbd OUT -> Cylinder In*)
2000, 4000, 6000:

	IF State = 4000 THEN
		DeltaP  := LS_P.Pos - CFG.TgtLS_P_Mid; 		(*Negative*)
		DeltaS  := LS_S.Pos - CFG.TgtLS_S_Mid; 		(*Positive*)
		DeltaPS := DeltaP + DeltaS + CFG.LS_Dif_Tgt;(*Positive -> Out Late*)

	ELSIF State = 6000 THEN
		DeltaP  := LS_P.Pos - CFG.TgtLS_P_OutR; 	(*Negative*)
		DeltaS  := LS_S.Pos - CFG.TgtLS_S_InR; 		(*Positive*)
		DeltaPS := DeltaP + DeltaS + CFG.LS_Dif_Tgt;(*Positive -> Out Late*)

	ELSIF Keel_Err OR Keel_Pos < CFG.Keel_S_Min THEN
		DeltaP  := LS_P.Pos - CFG.TgtLS_P_Safe_In; 	(*Negative*)
		DeltaS  := LS_S.Pos - CFG.TgtLS_S_Safe_Out; (*Positive*)
		DeltaPS := DeltaP + DeltaS + CFG.LS_Dif_Tgt;(*Positive -> Out Late*)

	ELSE
		DeltaP  := LS_P.Pos - CFG.TgtLS_P_In; 		(*Negative*)
		DeltaS  := LS_S.Pos - CFG.TgtLS_S_Out; 		(*Positive*)
		DeltaPS := DeltaP + DeltaS + CFG.LS_Dif_Tgt;(*Positive -> Out Late*)

	END_IF

	IF Hyst_Cnt > CFG.P_Hyst_TM THEN
		Hyst_ON := TRUE;
	ELSE
		Hyst_ON  := FALSE;
		Hyst_Cnt := Hyst_Cnt + CFG.Cycle;
	END_IF

	IF Manual OR NOT Ready OR SF_P.Alarm.Alarm OR LS_Err OR P_Alarm OR TimeOut THEN
		OUT_EVB_S := FALSE;
		OUT_EVT_S := FALSE;
		OUT_TWC_P := 0;
		OUT_TWC_S := 0;
		OUT_LP    := 0;
		State     := 0;

	ELSIF DeltaP >= 0.0 AND DeltaS <= 0.0 THEN
		OUT_EVB_S := FALSE;
		OUT_EVT_S := FALSE;
		OUT_TWC_P := 0;
		OUT_TWC_S := 0;
		OUT_LP    := 0;
		State     := 0;

	ELSE
		(*Activate SoftStop*)
		IF Event_P = INIT_CONTINUOUS OR Event_S = INIT_CONTINUOUS OR Event_C = INIT_CONTINUOUS
		OR State = 2000 AND ((NOT EngReady OR NOT Latching) AND Event_S = END_CONTINUOUS)
		OR State = 4000 AND ((NOT EngReady OR NOT Latching) AND Event_C = END_CONTINUOUS)
		OR State = 6000 AND ((NOT EngReady OR NOT Latching) AND Event_P = END_CONTINUOUS)
		THEN
			IF SoftStop THEN
				OUT_EVB_S := FALSE;
				OUT_EVT_S := FALSE;
				OUT_TWC_P := 0;
				OUT_TWC_S := 0;
				OUT_LP    := 0;
				State     := 0;
				RETURN;

			ELSE
				SoftStop := TRUE;

			END_IF
		END_IF

		(*Port IN  -> Cylinder Out*)
		IF SoftStop OR DeltaPS > CFG.LS_Dif_Min THEN
			TWC_P_Inc := TWC_P_Inc + CFG.EVP_In_Dec * CFG.Cycle; 						(*Increment*)
			TWC_P_Inc := MAX(TWC_P_Inc, -CFG.EVP_In_P_Max); 							(*Max Value*)
			TWC_P_Inc := MAX(TWC_P_Inc, -CFG.EVP_In_P_Min + DeltaP * CFG.EVP_In_LS_K); 	(*Approx K*)
			TWC_P_Inc := MIN(TWC_P_Inc, -CFG.EVP_In_P_Min); 							(*Min Value - Extra check*)

			IF TWC_P_Inc = -CFG.EVP_In_P_Min OR CFG.EVP_In_Dec <= 0
			THEN OUT_TWC_P := 0;
			ELSE OUT_TWC_P := REAL_TO_INT(TWC_P_Inc * 10.0);
			END_IF

		ELSIF DeltaP < 0.0 (*AND DeltaPS < CFG.LS_Dif_Min*) THEN
			TWC_P_Inc := TWC_P_Inc - CFG.EVP_In_Inc * CFG.Cycle; 						(*Increment*)
			TWC_P_Inc := MAX(TWC_P_Inc, -CFG.EVP_In_P_Max); 							(*Max Value*)
			TWC_P_Inc := MAX(TWC_P_Inc, -CFG.EVP_In_P_Min + DeltaP * CFG.EVP_In_LS_K); 	(*Approx K*)

			IF EngReady																	(*Delta K*)
			THEN TWC_P_Inc := MAX(TWC_P_Inc, -CFG.EVP_In_P_Eng + DeltaPS * CFG.EVP_In_EVP_K);
			ELSE TWC_P_Inc := MAX(TWC_P_Inc, -CFG.EVP_In_P_PP  + DeltaPS * CFG.EVP_In_EVP_K);
			END_IF

			TWC_P_Inc := MIN(TWC_P_Inc, -CFG.EVP_In_P_Min); 							(*Min Value - Extra check*)

			OUT_TWC_P := REAL_TO_INT(TWC_P_Inc * 10.0);

		ELSE
			OUT_TWC_P := 0;

		END_IF

		(*Stbd OUT -> Cylinder In*)
		IF SoftStop OR DeltaPS < -CFG.LS_Dif_Max THEN
			TWC_S_Inc := TWC_S_Inc - CFG.EVP_Out_Dec * CFG.Cycle; 						(*Increment*)
			TWC_S_Inc := MIN(TWC_S_Inc, CFG.EVP_Out_S_Max);								(*Max Value*)
			TWC_S_Inc := MIN(TWC_S_Inc, CFG.EVP_Out_S_Min + DeltaS * CFG.EVP_Out_LS_K); (*Approx K*)
			TWC_S_Inc := MAX(TWC_S_Inc, CFG.EVP_Out_S_Min); 							(*Min Value - Extra check*)

			IF TWC_S_Inc = CFG.EVP_Out_S_Min OR CFG.EVP_Out_Dec <= 0 THEN
				OUT_TWC_S := 0;
				OUT_EVB_S := FALSE;
			ELSE
				OUT_TWC_S := REAL_TO_INT(TWC_S_Inc * 10.0);
				OUT_EVB_S := TRUE;
			END_IF

			OUT_EVT_S := FALSE;

		ELSIF DeltaS > 0.0 (*AND DeltaPS > -CFG.LS_Dif_Max*) THEN
			TWC_S_Inc := TWC_S_Inc + CFG.EVP_Out_Inc * CFG.Cycle; 						(*Increment*)
			TWC_S_Inc := MIN(TWC_S_Inc, CFG.EVP_Out_S_Max);								(*Max Value*)
			TWC_S_Inc := MIN(TWC_S_Inc, CFG.EVP_Out_S_Min + DeltaS * CFG.EVP_Out_LS_K); (*Approx K*)

			IF EngReady																	(*Delta K*)
			THEN TWC_S_Inc := MIN(TWC_S_Inc, CFG.EVP_Out_S_Eng + DeltaPS * CFG.EVP_Out_EVP_K);
			ELSE TWC_S_Inc := MIN(TWC_S_Inc, CFG.EVP_Out_S_PP  + DeltaPS * CFG.EVP_Out_EVP_K);
			END_IF

			TWC_S_Inc := MAX(TWC_S_Inc, CFG.EVP_Out_S_Min); 							(*Min Value - Extra check*)

			OUT_TWC_S := REAL_TO_INT(TWC_S_Inc * 10.0);
			OUT_EVB_S := TRUE;

			IF Hyst_Cnt > CFG.P_Hyst_TM THEN
				Hyst_ON := TRUE;
			ELSE
				Hyst_ON  := FALSE;
				Hyst_Cnt := Hyst_Cnt + CFG.Cycle;
			END_IF
	
			IF PB_S.Bar > CFG.P_Hyst_HP AND Hyst_ON OR PB_S.Err THEN
				OUT_EVT_S := TRUE;
				Hyst_cnt  := 0.0;
			ELSIF PB_S.Bar < CFG.P_Hyst_LP AND Hyst_ON THEN
				OUT_EVT_S := FALSE;
				Hyst_cnt  := 0.0;
			END_IF

		ELSE
			OUT_TWC_S := 0;
			OUT_EVB_S := FALSE;
			OUT_EVT_S := FALSE;

		END_IF

		OUT_LP    := CFG.LP;

		(*If both stopped go to Init State*)
		IF OUT_TWC_P = 0 AND OUT_TWC_S = 0 THEN
			OUT_EVB_S := FALSE;
			OUT_EVT_S := FALSE;
			OUT_TWC_P := 0;
			OUT_TWC_S := 0;
			OUT_LP    := 0;
			State     := 0;

		END_IF

	END_IF

END_CASE
END_FUNCTION_BLOCK

(* POU FB/FB_KEEL, ST *)
FUNCTION_BLOCK FB_KEEL
VAR_INPUT
	Enable : BOOL;
	Ready  : BOOL;

	EngReady : BOOL;
	Latching : BOOL;

	AutoEase : BOOL;

	IN_I : ARRAY[1..4] OF BOOL;
	IN_O : ARRAY[1..4] OF BOOL;
	IN_C : ARRAY[1..4] OF BOOL;
	IN_F : ARRAY[1..4] OF BOOL;
	IN_T : ARRAY[1..2] OF BOOL;
END_VAR
VAR_IN_OUT
	LS_BOARD_P : ST_SENSOR_POS;
	LS_BOARD_S : ST_SENSOR_POS;

	P_I  : ST_SENSOR_BAR;
	P_O  : ST_SENSOR_BAR;
	LS1  : ST_SENSOR_POS;
	LS2  : ST_SENSOR_POS;

	CFG  : ST_KEEL_CFG;
END_VAR
VAR_OUTPUT
	EV_Eng_PI : BOOL;
	EV_Eng_EI : BOOL;
	EV_Eng_PO : BOOL;
	EV_Eng_EO : BOOL;
	EV_PP_I  : BOOL;
	EV_PP_O  : BOOL;

	EVP_Eng_I : UINT;
	EVP_Eng_O : UINT;

	EVP_SE_I  : UINT; (*mA*)
	EVP_SE_O  : UINT;
	EVP_FE_I  : UINT;
	EVP_FE_O  : UINT;

	P_Fill  : REAL; (*Bar*)
	P_Empty : REAL;

	EVP_Fill : INT; (*%*)

	OUT_LP   : BYTE;
END_VAR
VAR
	State   : WORD;

	IN_Hmi_I : BOOL;
	IN_Hmi_O : BOOL;
	IN_Hmi_C : BOOL;
	IN_Hmi_F : BOOL;
	IN_Hmi_T : BOOL;
	IN_Hmi_fill : BOOL;

	SI_I : ARRAY[1..5] OF FB_SMART_INPUT;
	SI_O : ARRAY[1..5] OF FB_SMART_INPUT;
	SI_C : ARRAY[1..5] OF FB_SMART_INPUT;
	SI_F : ARRAY[1..5] OF FB_SMART_INPUT;
	SI_T : ARRAY[1..3] OF FB_SMART_INPUT;

	SI_Hmi_fill : FB_SMART_INPUT;
	IN_Hmi_fill_Perc : INT := 20;

	Event_I : EN_SMART_INPUT_STATE;
	Event_O : EN_SMART_INPUT_STATE;
	Event_C : EN_SMART_INPUT_STATE;
	Event_F : EN_SMART_INPUT_STATE;
	Event_T : EN_SMART_INPUT_STATE;

	TimeCnt : REAL;
	TimeOut : BOOL;

	KEEL_I : BOOL;
	KEEL_SI : BOOL;
	KEEL_C : BOOL;
	KEEL_SO : BOOL;
	KEEL_O : BOOL;

	MOVING_I : BOOL;
	MOVING_O : BOOL;
	MOVING_C : BOOL;
	MOVING_F : BOOL;
	MOVING_T : BOOL;

	EnableFill : BOOL;
	BypassSF   : BOOL;

	P_Alarm: BOOL;
	LS_Pos : REAL;
	LS_Err : BOOL;

	EVP_In_SE_Tgt  : REAL; (*mA*)
	EVP_In_FE_Tgt  : REAL;
	EVP_Out_SE_Tgt : REAL;
	EVP_Out_FE_Tgt : REAL;

	EVP_In_Eng_Tgt  : REAL;
	EVP_Out_Eng_Tgt : REAL;

	EVP_Out_Fill_Tgt : REAL;

	TgtLS   : REAL;
	DeltaLS : REAL;

	(*Anadir alrmas al keel*)
	SoftStop: BOOL;
END_VAR
VAR PERSISTENT
	Manual AT %Q*: BOOL;
END_VAR
(*
IN  = keel to STBD
OUT = Keel to PORT
*)

P_Alarm := P_I.AlMax OR P_O.AlMax;

(*Evaluo los LS1 y LS2*)
IF NOT LS1.Err THEN
	LS_Pos := LS1.Pos;
	LS_Err := FALSE;
ELSIF NOT LS2.Err THEN
	LS_Pos := LS2.Pos;
	LS_Err := FALSE;
ELSE
	LS_Pos := 0;
	LS_Err := TRUE;
END_IF

KEEL_I := NOT LS_Err AND LS_Pos < CFG.TgtLS_In  + CFG.LS_DB;
KEEL_O := NOT LS_Err AND LS_Pos > CFG.TgtLS_Out - CFG.LS_DB;

KEEL_SI := NOT LS_Err AND LS_Pos < CFG.TgtLS_Safe_In  + CFG.LS_DB;
KEEL_SO := NOT LS_Err AND LS_Pos > CFG.TgtLS_Safe_Out - CFG.LS_DB;

KEEL_C := NOT LS_Err AND CFG.LS_DB > ABS(CFG.TgtLS_Mid - LS_Pos);

(*Check Inputs*)
SI_I[1](In:= IN_I[1],  T_Cont:= T#0ms, T_DClk:= T#0ms);
SI_I[2](In:= IN_I[2],  T_Cont:= T#0ms, T_DClk:= T#0ms);
SI_I[3](In:= IN_I[3],  T_Cont:= T#0ms, T_DClk:= T#0ms);
SI_I[4](In:= IN_I[4],  T_Cont:= T#0ms, T_DClk:= T#0ms);
SI_I[5](In:= IN_Hmi_I, T_Cont:= T#0ms, T_DClk:= T#0ms);

SI_O[1](In:= IN_O[1],  T_Cont:= T#0ms, T_DClk:= T#0ms);
SI_O[2](In:= IN_O[2],  T_Cont:= T#0ms, T_DClk:= T#0ms);
SI_O[3](In:= IN_O[3],  T_Cont:= T#0ms, T_DClk:= T#0ms);
SI_O[4](In:= IN_O[4],  T_Cont:= T#0ms, T_DClk:= T#0ms);
SI_O[5](In:= IN_Hmi_O, T_Cont:= T#0ms, T_DClk:= T#0ms);

SI_C[1](In:= IN_C[1],  T_Cont:= T#0ms, T_DClk:= T#0ms);
SI_C[2](In:= IN_C[2],  T_Cont:= T#0ms, T_DClk:= T#0ms);
SI_C[3](In:= IN_C[3],  T_Cont:= T#0ms, T_DClk:= T#0ms);
SI_C[4](In:= IN_C[4],  T_Cont:= T#0ms, T_DClk:= T#0ms);
SI_C[5](In:= IN_Hmi_C, T_Cont:= T#0ms, T_DClk:= T#0ms);

SI_F[1](In:= IN_F[1],  T_Cont:= T#0ms, T_DClk:= T#0ms);
SI_F[2](In:= IN_F[2],  T_Cont:= T#0ms, T_DClk:= T#0ms);
SI_F[3](In:= IN_F[3],  T_Cont:= T#0ms, T_DClk:= T#0ms);
SI_F[4](In:= IN_F[4],  T_Cont:= T#0ms, T_DClk:= T#0ms);
SI_F[5](In:= IN_Hmi_F, T_Cont:= T#0ms, T_DClk:= T#0ms);

SI_T[1](In:= IN_T[1],  T_Cont:= T#0ms, T_DClk:= T#0ms);
SI_T[2](In:= IN_T[2],  T_Cont:= T#0ms, T_DClk:= T#0ms);
SI_T[3](In:= IN_Hmi_T, T_Cont:= T#0ms, T_DClk:= T#0ms);

SI_Hmi_fill(In:= IN_Hmi_fill, T_Cont:= T#0ms, T_DClk:= T#0ms);

IF NOT Enable THEN
	EV_Eng_PI := FALSE;
	EV_Eng_EI := FALSE;
	EV_Eng_PO := FALSE;
	EV_Eng_EO := FALSE;
	EV_PP_I  := FALSE;
	EV_PP_O  := FALSE;

	EVP_Eng_I := 0; (*mA*)
	EVP_Eng_O := 0;

	EVP_FE_I  := 0;
	EVP_FE_O  := 0;
	EVP_SE_I  := 0; (*mA*)
	EVP_SE_O  := 0;

	P_Fill  := 0; (*bar*)
	P_Empty := 0;

	EVP_Fill := 0; (*%*)

	OUT_LP  := 0;

	EnableFill := FALSE;

	TimeCnt := 0.0;
	State   := 0;
	RETURN;
END_IF

IF NOT Manual THEN
	EnableFill := FALSE;
	BypassSF   := FALSE;
END_IF

(*Check Time*)
TimeOut := TimeOut OR ( CFG.TimeMax > 0  AND TimeCnt > CFG.TimeMax );
TimeCnt := TimeCnt + CFG.Cycle;

IF    SI_I[1].Event <> NONE THEN Event_I := SI_I[1].Event;
ELSIF SI_I[2].Event <> NONE THEN Event_I := SI_I[2].Event;
ELSIF SI_I[3].Event <> NONE THEN Event_I := SI_I[3].Event;
ELSIF SI_I[4].Event <> NONE THEN Event_I := SI_I[4].Event;
ELSIF SI_I[5].Event <> NONE THEN Event_I := SI_I[5].Event;
ELSE
	Event_I := NONE;
END_IF

IF    SI_O[1].Event <> NONE THEN Event_O := SI_O[1].Event;
ELSIF SI_O[2].Event <> NONE THEN Event_O := SI_O[2].Event;
ELSIF SI_O[3].Event <> NONE THEN Event_O := SI_O[3].Event;
ELSIF SI_O[4].Event <> NONE THEN Event_O := SI_O[4].Event;
ELSIF SI_O[5].Event <> NONE THEN Event_O := SI_O[5].Event;
ELSE
	Event_O := NONE;
END_IF

IF    SI_C[1].Event <> NONE THEN Event_C := SI_C[1].Event;
ELSIF SI_C[2].Event <> NONE THEN Event_C := SI_C[2].Event;
ELSIF SI_C[3].Event <> NONE THEN Event_C := SI_C[3].Event;
ELSIF SI_C[4].Event <> NONE THEN Event_C := SI_C[4].Event;
ELSIF SI_C[5].Event <> NONE THEN Event_C := SI_C[5].Event;
ELSE
	Event_C := NONE;
END_IF

IF    SI_F[1].Event <> NONE THEN Event_F := SI_F[1].Event;
ELSIF SI_F[2].Event <> NONE THEN Event_F := SI_F[2].Event;
ELSIF SI_F[3].Event <> NONE THEN Event_F := SI_F[3].Event;
ELSIF SI_F[4].Event <> NONE THEN Event_F := SI_F[4].Event;
ELSIF SI_F[5].Event <> NONE THEN Event_F := SI_F[5].Event;
ELSE
	Event_F := NONE;
END_IF

IF    SI_T[1].Event <> NONE THEN Event_T := SI_T[1].Event;
ELSIF SI_T[2].Event <> NONE THEN Event_T := SI_T[2].Event;
ELSIF SI_T[3].Event <> NONE THEN Event_T := SI_T[3].Event;
ELSE
	Event_T := NONE;
END_IF

(*Working States*)
CASE State OF

(*Init State*)
0:
	EV_Eng_PI := FALSE;
	EV_Eng_EI := FALSE;
	EV_Eng_PO := FALSE;
	EV_Eng_EO := FALSE;
	EV_PP_I   := FALSE;
	EV_PP_O   := FALSE;
	EVP_Eng_I := 0; (*mA*)
	EVP_Eng_O := 0;
	EVP_SE_I := 0; (*mA*)
	EVP_SE_O := 0;
	EVP_FE_I := 0;
	EVP_FE_O := 0;
	P_Fill   := 0; (*bar*)
	P_Empty  := 0;
	EVP_Fill := 0; (*%*)
	OUT_LP   := 0;

	TimeCnt  := 0.0;

	MOVING_I := FALSE;
	MOVING_O := FALSE;
	MOVING_C := FALSE;
	MOVING_F := FALSE;

	SoftStop := FALSE;

	(*Start IN*)
	IF Event_I = INIT_CONTINUOUS AND Ready AND NOT P_I.AlMax THEN
		TimeOut  := FALSE;
		MOVING_I := TRUE;

		(*Next State*)
		IF Manual (*OR LS_Err*) THEN
			State := 100;
		ELSE
			TgtLS := CFG.TgtLS_In;
			State := 1000;
		END_IF

		EVP_In_Eng_Tgt := CFG.EVP_In_Eng_Min;

	(*Start OUT*)
	ELSIF Event_O = INIT_CONTINUOUS AND Ready AND NOT P_O.AlMax THEN
		TimeOut  := FALSE;
		MOVING_O := TRUE;

		(*Next State*)
		IF Manual (*OR LS_Err*) THEN
			State := 200;
		ELSE
			TgtLS := CFG.TgtLS_OUT;
			State := 2000;
		END_IF

		EVP_Out_Eng_Tgt := CFG.EVP_Out_Eng_Min;

	(*Start CENTER*)
	ELSIF Event_C = INIT_CONTINUOUS AND Ready AND NOT LS_Err AND NOT Manual AND NOT KEEL_C THEN
		TimeOut  := FALSE;
		MOVING_C := TRUE;

		IF LS_Pos > CFG.TgtLS_Mid AND NOT P_I.AlMax THEN
			MOVING_I := TRUE;
			TgtLS    := CFG.TgtLS_Mid;
			State    := 1100;  (*Next State*)

			EVP_In_Eng_Tgt := CFG.EVP_In_Eng_Min;

		ELSIF LS_Pos < CFG.TgtLS_Mid AND NOT P_O.AlMax THEN
			MOVING_O := TRUE;
			TgtLS    := CFG.TgtLS_Mid;
			State    := 2100;  (*Next State*)

			EVP_Out_Eng_Tgt := CFG.EVP_Out_Eng_Min;

		END_IF

	(*Start Tack*)
	ELSIF Event_T = INIT_CONTINUOUS AND EngReady AND Latching AND Ready AND NOT LS_Err AND NOT Manual AND NOT KEEL_C THEN
		TimeOut  := FALSE;
		MOVING_T := TRUE;

		IF LS_Pos + CFG.TgtLS_Tack_Off > CFG.TgtLS_Mid AND NOT P_I.AlMax THEN
			MOVING_I := TRUE;
			TgtLS    := CFG.TgtLS_In + CFG.TgtLS_Out - LS_Pos - CFG.TgtLS_Tack_Off;
			State    := 1200;  (*Next State*)

			EVP_In_Eng_Tgt := CFG.EVP_In_Eng_Min;

		ELSIF LS_Pos - CFG.TgtLS_Tack_Off < CFG.TgtLS_Mid AND NOT P_O.AlMax THEN
			MOVING_O := TRUE;
			TgtLS    := CFG.TgtLS_Out + CFG.TgtLS_In - LS_Pos + CFG.TgtLS_Tack_Off;
			State    := 2200;  (*Next State*)

			EVP_Out_Eng_Tgt := CFG.EVP_Out_Eng_Min;

		END_IF

	(*Start FLOAT*)
	ELSIF Event_F = INIT_CONTINUOUS AND Ready THEN
		TimeOut  := FALSE;
		MOVING_F := TRUE;

		IF Manual (*OR LS_Err*)  THEN
			State := 300;

			EVP_In_SE_Tgt := CFG.EVP_In_SE_Min;
			EVP_In_FE_Tgt := CFG.EVP_In_FE_Min;
			EVP_Out_SE_Tgt := CFG.EVP_Out_SE_Min;
			EVP_Out_FE_Tgt := CFG.EVP_Out_FE_Min;

		ELSE
			IF LS_Pos > CFG.TgtLS_Mid + CFG.LS_DB AND P_O.Bar > P_I.Bar THEN (*Ease Out, Then Moving In*)
				State := 3000;

				EVP_Out_SE_Tgt := CFG.EVP_Out_SE_Min;
				EVP_Out_FE_Tgt := CFG.EVP_Out_FE_Min;

			ELSIF LS_Pos < CFG.TgtLS_Mid - CFG.LS_DB AND P_I.Bar > P_O.Bar THEN (*Ease In, Then Moving Out*)
				State := 4000;

				EVP_In_SE_Tgt := CFG.EVP_In_SE_Min;
				EVP_In_FE_Tgt := CFG.EVP_In_FE_Min;

			END_IF
		END_IF

	(*Start Fill*)
	ELSIF SI_Hmi_fill.Event = INIT_CONTINUOUS AND Manual AND EnableFill THEN
		TimeOut := FALSE;
		State   := 500;

	(*Auto Ease*)
	ELSIF AutoEase THEN
		(*On Port - Cyl Out, Release IN*)
		IF KEEL_SO AND P_O.Bar > CFG.MinLoadSide_Bar AND P_I.Bar > CFG.MaxUnloadSide_Bar THEN
			EVP_SE_I := REAL_TO_UINT( CFG.EVP_In_SE_Man );

		(*On Stbd - Cyl In, Release OUT*)
		ELSIF KEEL_SI AND P_I.Bar > CFG.MinLoadSide_Bar AND P_O.Bar > CFG.MaxUnloadSide_Bar THEN
			EVP_SE_O := REAL_TO_UINT( CFG.EVP_Out_SE_Man );

		END_IF

	END_IF

(*Manual IN*)
100:
	IF TimeOut OR P_I.AlMax THEN
		Out_LP := 0;
		State  := 0;  (*Next State*)

	ELSIF EngReady THEN
		(*Activate SoftStop*)
		IF Event_I <> NONE
		OR Event_O = INIT_CONTINUOUS
		OR Event_C = INIT_CONTINUOUS
		OR Event_F = INIT_CONTINUOUS
		OR Event_T = INIT_CONTINUOUS
		THEN
			(*If already stoping, full stop*)
			IF SoftStop THEN
				OUT_LP   := 0;
				State    := 0; (*Next State*)
				RETURN;

			ELSE
				SoftStop := TRUE;

			END_IF
		END_IF

		IF SoftStop THEN
			EVP_In_Eng_Tgt := EVP_In_Eng_Tgt - CFG.EVP_In_Eng_Dec * CFG.Cycle;
			EVP_In_Eng_Tgt := MIN(EVP_In_Eng_Tgt, CFG.EVP_In_Eng_Max);
			EVP_In_Eng_Tgt := MIN(EVP_In_Eng_Tgt, CFG.EVP_In_Eng_Man);
			EVP_In_Eng_Tgt := MAX(EVP_In_Eng_Tgt, CFG.EVP_In_Eng_Min);

			IF EVP_In_Eng_Tgt = CFG.EVP_In_Eng_Min OR CFG.EVP_In_Eng_Dec <= 0
			THEN EVP_Eng_I := 0;
			ELSE EVP_Eng_I := REAL_TO_UINT(EVP_In_Eng_Tgt);
			END_IF

		ELSE
			EVP_In_Eng_Tgt := EVP_In_Eng_Tgt + CFG.EVP_In_Eng_Inc * CFG.Cycle;
			EVP_In_Eng_Tgt := MIN(EVP_In_Eng_Tgt, CFG.EVP_In_Eng_Max);
			EVP_In_Eng_Tgt := MIN(EVP_In_Eng_Tgt, CFG.EVP_In_Eng_Man);
			EVP_In_Eng_Tgt := MAX(EVP_In_Eng_Tgt, CFG.EVP_In_Eng_Min);

			EVP_Eng_I := REAL_TO_UINT(EVP_In_Eng_Tgt);

		END_IF

		IF EVP_Eng_I = 0 THEN
			OUT_LP   := 0;
			State    := 0; (*Next State*)

		ELSE
			EV_Eng_PI := TRUE;
			EV_Eng_EO := TRUE;
			EV_PP_I   := FALSE;
		(*	EVP_Eng_I*)
			EVP_SE_O  := REAL_TO_UINT(CFG.EVP_Out_SE_Empty);
			P_Empty   := CFG.EVP_In_P_Empty; (*bar*)
			OUT_LP    := 1;

		END_IF

	ELSE
		IF Event_I <> NONE
		OR Event_O = INIT_CONTINUOUS
		OR Event_C = INIT_CONTINUOUS
		OR Event_F = INIT_CONTINUOUS
		OR Event_T = INIT_CONTINUOUS
		THEN
			OUT_LP   := 0;
			State    := 0; (*Next State*)

		ELSE
			EV_Eng_PI := FALSE;
			EV_Eng_EO := FALSE;
			EV_PP_I   := TRUE;
			EVP_Eng_I := 0; (*mA*)
			EVP_SE_O  := 0;
			P_Empty   := 0;
			OUT_LP    := 1;

		END_IF
	END_IF

(*Manual out*)
200:
	IF TimeOut OR P_O.AlMax THEN
		Out_LP := 0;
		State  := 0;  (*Next State*)

	ELSIF EngReady THEN

		IF Event_I = INIT_CONTINUOUS
		OR Event_O <> NONE
		OR Event_C = INIT_CONTINUOUS
		OR Event_F = INIT_CONTINUOUS
		OR Event_T = INIT_CONTINUOUS
		THEN
			(*If already stoping, full stop*)
			IF SoftStop THEN
				OUT_LP   := 0;
				State    := 0; (*Next State*)
				RETURN;

			ELSE
				SoftStop := TRUE;

			END_IF
		END_IF

		IF SoftStop THEN
			EVP_Out_Eng_Tgt := EVP_Out_Eng_Tgt - CFG.EVP_Out_Eng_Dec * CFG.Cycle;
			EVP_Out_Eng_Tgt := MIN(EVP_Out_Eng_Tgt, CFG.EVP_Out_Eng_Max);
			EVP_Out_Eng_Tgt := MIN(EVP_Out_Eng_Tgt, CFG.EVP_Out_Eng_Man);
			EVP_Out_Eng_Tgt := MAX(EVP_Out_Eng_Tgt, CFG.EVP_Out_Eng_Min);

			IF EVP_Out_Eng_Tgt = CFG.EVP_Out_Eng_Min OR CFG.EVP_Out_Eng_Dec <= 0
			THEN EVP_Eng_O := 0;
			ELSE EVP_Eng_O := REAL_TO_UINT(EVP_Out_Eng_Tgt);
			END_IF

		ELSE
			EVP_Out_Eng_Tgt := EVP_Out_Eng_Tgt + CFG.EVP_Out_Eng_Inc * CFG.Cycle;
			EVP_Out_Eng_Tgt := MIN(EVP_Out_Eng_Tgt, CFG.EVP_Out_Eng_Max);
			EVP_Out_Eng_Tgt := MIN(EVP_Out_Eng_Tgt, CFG.EVP_Out_Eng_Man);
			EVP_Out_Eng_Tgt := MAX(EVP_Out_Eng_Tgt, CFG.EVP_Out_Eng_Min);

			EVP_Eng_O := REAL_TO_UINT(EVP_Out_Eng_Tgt);

		END_IF

		IF EVP_Eng_O = 0 THEN
			OUT_LP   := 0;
			State    := 0; (*Next State*)

		ELSE
			EVP_Out_Fill_Tgt := EVP_Out_Eng_Tgt * CFG.EVP_Out_Fill_K + CFg.EVP_Out_Fill_Off;
			EVP_Out_Fill_Tgt := MIN(EVP_Out_Fill_Tgt, CFG.EVP_Out_Fill_Max);
			EVP_Out_Fill_Tgt := MAX(EVP_Out_Fill_Tgt, CFG.EVP_Out_Fill_Min);
	
			EV_Eng_EI := TRUE;
			EV_Eng_PO := TRUE;
			EV_PP_O   := FALSE;
		(*	EVP_Eng_O*)
			P_Fill    := CFG.EVP_Out_P_Fill; (*bar*)
			EVP_Fill  := REAL_TO_INT(EVP_Out_Fill_Tgt * 10.0); (*%*)
			OUT_LP    := 1;

		END_IF

	ELSE
		IF Event_I = INIT_CONTINUOUS
		OR Event_O <> NONE
		OR Event_C = INIT_CONTINUOUS
		OR Event_F = INIT_CONTINUOUS
		OR Event_T = INIT_CONTINUOUS
		THEN
			OUT_LP   := 0;
			State    := 0; (*Next State*)

		ELSE
			EV_Eng_EI := FALSE;
			EV_Eng_PO := FALSE;
			EV_PP_O   := TRUE;
			EVP_Eng_O := 0;  (*mA*)
			P_Fill    := 0; (*bar*)
			EVP_Fill  := 0; (*%*)
			OUT_LP    := 1;

		END_IF
	END_IF

(*Manual FLOAT*)
300:
	IF TimeOut THEN
		Out_LP := 0;
		State  := 0;  (*Next State*)

	ELSE
		(*Activate SoftStop*)
		IF Event_F <> NONE
		OR Event_I = INIT_CONTINUOUS
		OR Event_C = INIT_CONTINUOUS
		OR Event_O = INIT_CONTINUOUS
		OR Event_T = INIT_CONTINUOUS
		THEN

			(*If already stoping, full stop*)
			IF SoftStop THEN
				OUT_LP    := 0;
				State     := 0; (*Next State*)
				RETURN;

			ELSE
				SoftStop := TRUE;

			END_IF
		END_IF

		IF SoftStop THEN
			EVP_In_FE_Tgt := EVP_In_FE_Tgt - CFG.EVP_In_FE_Dec * CFG.Cycle;
			EVP_In_FE_Tgt := MIN(EVP_In_FE_Tgt, CFG.EVP_In_FE_Max);
			EVP_In_FE_Tgt := MIN(EVP_In_FE_Tgt, CFG.EVP_In_FE_Man);
			EVP_In_FE_Tgt := MAX(EVP_In_FE_Tgt, CFG.EVP_In_FE_Min);

			EVP_Out_FE_Tgt := EVP_Out_FE_Tgt - CFG.EVP_Out_FE_Dec * CFG.Cycle;
			EVP_Out_FE_Tgt := MIN(EVP_Out_FE_Tgt, CFG.EVP_Out_FE_Max);
			EVP_Out_FE_Tgt := MIN(EVP_Out_FE_Tgt, CFG.EVP_Out_FE_Man);
			EVP_Out_FE_Tgt := MAX(EVP_Out_FE_Tgt, CFG.EVP_Out_FE_Min);

			IF EVP_In_FE_Tgt = CFG.EVP_In_FE_Min THEN
				EVP_In_SE_Tgt := EVP_In_SE_Tgt - CFG.EVP_In_SE_Dec * CFG.Cycle;
				EVP_In_SE_Tgt := MIN(EVP_In_SE_Tgt, CFG.EVP_In_SE_Max);
				EVP_In_SE_Tgt := MIN(EVP_In_SE_Tgt, CFG.EVP_In_SE_Man);
				EVP_In_SE_Tgt := MAX(EVP_In_SE_Tgt, CFG.EVP_In_SE_Min);
			END_IF

			IF EVP_Out_FE_Tgt = CFG.EVP_Out_FE_Min THEN
				EVP_Out_SE_Tgt := EVP_Out_SE_Tgt - CFG.EVP_Out_SE_Dec * CFG.Cycle;
				EVP_Out_SE_Tgt := MIN(EVP_Out_SE_Tgt, CFG.EVP_Out_SE_Max);
				EVP_Out_SE_Tgt := MIN(EVP_Out_SE_Tgt, CFG.EVP_Out_SE_Man);
				EVP_Out_SE_Tgt := MAX(EVP_Out_SE_Tgt, CFG.EVP_Out_SE_Min);
			END_IF


			IF EVP_In_SE_Tgt = CFG.EVP_In_SE_Min OR CFG.EVP_In_SE_Dec <= 0
			THEN EVP_SE_I := 0;
			ELSE EVP_SE_I := REAL_TO_UINT(EVP_In_SE_Tgt );
			END_IF

			IF EVP_Out_SE_Tgt = CFG.EVP_Out_SE_Min OR CFG.EVP_Out_SE_Dec <= 0
			THEN EVP_SE_O := 0;
			ELSE EVP_SE_O := REAL_TO_UINT(EVP_Out_SE_Tgt );
			END_IF

			IF EVP_In_FE_Tgt = CFG.EVP_In_FE_Min OR CFG.EVP_In_FE_Dec <= 0
			THEN EVP_FE_I := 0;
			ELSE EVP_FE_I := REAL_TO_UINT(EVP_In_FE_Tgt );
			END_IF

			IF EVP_Out_FE_Tgt = CFG.EVP_Out_FE_Min OR CFG.EVP_Out_FE_Dec <= 0
			THEN EVP_FE_O := 0;
			ELSE EVP_FE_O := REAL_TO_UINT(EVP_Out_FE_Tgt );
			END_IF

		ELSE
			EVP_In_SE_Tgt := EVP_In_SE_Tgt + CFG.EVP_In_SE_Inc * CFG.Cycle;
			EVP_In_SE_Tgt := MIN(EVP_In_SE_Tgt, CFG.EVP_In_SE_Max);
			EVP_In_SE_Tgt := MIN(EVP_In_SE_Tgt, CFG.EVP_In_SE_Man);
			EVP_In_SE_Tgt := MAX(EVP_In_SE_Tgt, CFG.EVP_In_SE_Min);
	
			EVP_Out_SE_Tgt := EVP_Out_SE_Tgt + CFG.EVP_Out_SE_Inc * CFG.Cycle;
			EVP_Out_SE_Tgt := MIN(EVP_Out_SE_Tgt, CFG.EVP_Out_SE_Max);
			EVP_Out_SE_Tgt := MIN(EVP_Out_SE_Tgt, CFG.EVP_Out_SE_Man);
			EVP_Out_SE_Tgt := MAX(EVP_Out_SE_Tgt, CFG.EVP_Out_SE_Min);

			IF EVP_In_SE_Tgt = CFG.EVP_In_SE_Man OR EVP_In_SE_Tgt = CFG.EVP_In_SE_Max THEN
				EVP_In_FE_Tgt := EVP_In_FE_Tgt + CFG.EVP_In_FE_Inc * CFG.Cycle;
				EVP_In_FE_Tgt := MIN(EVP_In_FE_Tgt, CFG.EVP_In_FE_Max);
				EVP_In_FE_Tgt := MIN(EVP_In_FE_Tgt, CFG.EVP_In_FE_Man);
				EVP_In_FE_Tgt := MAX(EVP_In_FE_Tgt, CFG.EVP_In_FE_Min);
			END_IF
	
			IF EVP_Out_SE_Tgt = CFG.EVP_Out_SE_Man OR EVP_Out_SE_Tgt = CFG.EVP_Out_SE_Max THEN
				EVP_Out_FE_Tgt := EVP_Out_FE_Tgt + CFG.EVP_Out_FE_Inc * CFG.Cycle;
				EVP_Out_FE_Tgt := MIN(EVP_Out_FE_Tgt, CFG.EVP_Out_FE_Max);
				EVP_Out_FE_Tgt := MIN(EVP_Out_FE_Tgt, CFG.EVP_Out_FE_Man);
				EVP_Out_FE_Tgt := MAX(EVP_Out_FE_Tgt, CFG.EVP_Out_FE_Min);
			END_IF

			EVP_SE_I  := REAL_TO_UINT(EVP_In_SE_Tgt );
			EVP_SE_O  := REAL_TO_UINT(EVP_Out_SE_Tgt);
			EVP_FE_I  := REAL_TO_UINT(EVP_In_FE_Tgt );
			EVP_FE_O  := REAL_TO_UINT(EVP_Out_FE_Tgt);

		END_IF

		(*If ALL stopped go to Init State*)
		IF EVP_SE_I = 0 AND EVP_SE_O = 0 AND EVP_FE_I = 0 AND EVP_FE_O = 0 THEN
			Out_LP := 0;
			State  := 0;  (*Next State*)

		END_IF
	END_IF

(*Manual Fill*)
500:
	IF SI_Hmi_fill.Event = END_CONTINUOUS OR TimeOut OR NOT Manual OR NOT EnableFill THEN
		Out_LP := 0;
		State  := 0;  (*Next State*)

	ELSE
		EV_Eng_PI := FALSE;
		EV_Eng_EI := FALSE;
		EV_Eng_PO := FALSE;
		EV_Eng_EO := FALSE;
		EV_PP_I   := FALSE;
		EV_PP_O   := FALSE;
		EVP_Eng_I := 0; (*mA*)
		EVP_Eng_O := 0;
		EVP_SE_I  := 0;
		EVP_SE_O  := 0;
		EVP_FE_I  := 0;
		EVP_FE_O  := 0;
		P_Fill    := 0; (*bar*)
		P_Empty   := 0;
		EVP_Fill  := REAL_TO_INT(IN_Hmi_fill_Perc * 10.0); (*%*)
		OUT_LP    := 1;

	END_IF

(*Auto IN*)
1000,1100,1200:
	IF TgtLS < CFG.TgtLS_Safe_In AND (LS_BOARD_S.Err OR LS_BOARD_S.Pos < CFG.Board_S_Min_Out) THEN
		DeltaLS := LS_Pos - CFG.TgtLS_Safe_In; 			(*Positive*)

	ELSE
		DeltaLS := LS_Pos - MAX(TgtLS, CFG.TgtLS_In); 	(*Positive*)

	END_IF

	IF Manual OR NOT Ready OR LS_Err OR P_Alarm OR TimeOut THEN
		EV_Eng_PI := FALSE;
		EV_Eng_EO := FALSE;
		EV_PP_I   := FALSE;
		EVP_Eng_I := 0; (*mA*)
		EVP_SE_O  := 0;
		P_Empty   := 0; (*bar*)
		Out_LP    := 0;
		State     := 0; (*Next State*)

	ELSIF DeltaLS <= 0.0 THEN
		EV_Eng_PI := FALSE;
		EV_Eng_EO := FALSE;
		EV_PP_I   := FALSE;
		EVP_Eng_I := 0; (*mA*)
		EVP_SE_O  := 0;
		P_Empty   := 0;	(*bar*)
		Out_LP    := 0;
		State     := 0; (*Next State*)

	ELSIF EngReady THEN
		(*Activate SoftStop*)
		IF Event_I = INIT_CONTINUOUS OR State = 1000 AND NOT Latching AND Event_I = END_CONTINUOUS
		OR Event_O = INIT_CONTINUOUS
		OR Event_C = INIT_CONTINUOUS OR State = 1100 AND NOT Latching AND Event_C = END_CONTINUOUS
		OR Event_F = INIT_CONTINUOUS
		OR Event_T = INIT_CONTINUOUS OR State = 1200 AND NOT Latching AND Event_T = END_CONTINUOUS
		THEN
			(*If already stoping, full stop*)
			IF SoftStop THEN
				OUT_LP   := 0;
				State    := 0; (*Next State*)
				RETURN;

			ELSE
				SoftStop := TRUE;

			END_IF
		END_IF

		IF SoftStop THEN
			EVP_In_Eng_Tgt := EVP_In_Eng_Tgt - CFG.EVP_In_Eng_Dec * CFG.Cycle;
			EVP_In_Eng_Tgt := MIN(EVP_In_Eng_Tgt, CFG.EVP_In_Eng_Max);
			EVP_In_Eng_Tgt := MIN(EVP_In_Eng_Tgt, CFG.EVP_In_Eng_Min + DeltaLS * CFG.EVP_In_Eng_K);
			EVP_In_Eng_Tgt := MAX(EVP_In_Eng_Tgt, CFG.EVP_In_Eng_Min);

			IF EVP_In_Eng_Tgt = CFG.EVP_In_Eng_Min OR CFG.EVP_In_Eng_Dec <= 0
			THEN EVP_Eng_I := 0;
			ELSE EVP_Eng_I := REAL_TO_UINT(EVP_In_Eng_Tgt);
			END_IF

		ELSE
			EVP_In_Eng_Tgt := EVP_In_Eng_Tgt + CFG.EVP_In_Eng_Inc * CFG.Cycle;
			EVP_In_Eng_Tgt := MIN(EVP_In_Eng_Tgt, CFG.EVP_In_Eng_Max);
			EVP_In_Eng_Tgt := MIN(EVP_In_Eng_Tgt, CFG.EVP_In_Eng_Min + DeltaLS * CFG.EVP_In_Eng_K);
			EVP_In_Eng_Tgt := MAX(EVP_In_Eng_Tgt, CFG.EVP_In_Eng_Min);

			EVP_Eng_I := REAL_TO_UINT(EVP_In_Eng_Tgt);

		END_IF

		IF EVP_Eng_I = 0 THEN
			OUT_LP   := 0;
			State    := 0; (*Next State*)

		ELSE
			EV_Eng_PI := TRUE;
			EV_Eng_EO := TRUE;
			EV_PP_I   := FALSE;
		(*	EVP_Eng_I*)
			EVP_SE_O  := REAL_TO_UINT(CFG.EVP_Out_SE_Empty);
			P_Empty   := CFG.EVP_In_P_Empty; (*bar*)
			OUT_LP    := 1;

		END_IF

	ELSE
		IF Event_I = INIT_CONTINUOUS OR State = 1000 AND Event_I = END_CONTINUOUS
		OR Event_O = INIT_CONTINUOUS
		OR Event_C = INIT_CONTINUOUS OR State = 1100 AND Event_C = END_CONTINUOUS
		OR Event_F = INIT_CONTINUOUS
		OR Event_T = INIT_CONTINUOUS OR State = 1200 AND Event_T = END_CONTINUOUS
		THEN
			OUT_LP   := 0;
			State    := 0; (*Next State*)

		ELSE
			EV_Eng_PI := FALSE;
			EV_Eng_EO := FALSE;
			EV_PP_I   := TRUE;
			EVP_Eng_I := 0; (*mA*)
			EVP_SE_O  := 0;
			P_Empty   := 0;
			OUT_LP    := 1;

		END_IF
	END_IF

(*Auto OUT*)
2000,2100,2200:
	IF TgtLS > CFG.TgtLS_Safe_Out AND (LS_BOARD_P.Err OR LS_BOARD_P.Pos < CFG.Board_P_Min_Out) THEN
		DeltaLS := LS_Pos - CFG.TgtLS_Safe_Out; 		(*Negative*)

	ELSE
		DeltaLS := LS_Pos - MIN(TgtLS, CFG.TgtLS_Out); 	(*Negative*)

	END_IF

	IF Manual OR NOT Ready OR LS_Err OR P_Alarm OR TimeOut THEN
		EV_Eng_EI := FALSE;
		EV_Eng_PO := FALSE;
		EV_PP_O   := FALSE;
		EVP_Eng_O := 0; (*mA*)
		P_Fill    := 0; (*bar*)
		EVP_Fill  := 0; (*%*)
		OUT_LP    := 0;
		State     := 0; (*Next State*)

	ELSIF DeltaLS >= 0.0 THEN
		EV_Eng_EI := FALSE;
		EV_Eng_PO := FALSE;
		EV_PP_O   := FALSE;
		EVP_Eng_O := 0; (*mA*)
		P_Fill    := 0; (*bar*)
		EVP_Fill  := 0; (*%*)
		OUT_LP    := 0;
		State     := 0; (*Next State*)

	ELSIF EngReady THEN
		(*Activate SoftStop*)
		IF Event_I = INIT_CONTINUOUS
		OR Event_O = INIT_CONTINUOUS OR State = 2000 AND NOT Latching AND Event_O = END_CONTINUOUS
		OR Event_C = INIT_CONTINUOUS OR State = 2100 AND NOT Latching AND Event_C = END_CONTINUOUS
		OR Event_F = INIT_CONTINUOUS
		OR Event_T = INIT_CONTINUOUS OR State = 2200 AND NOT Latching AND Event_T = END_CONTINUOUS
		THEN
			(*If already stoping, full stop*)
			IF SoftStop THEN
				OUT_LP   := 0;
				State    := 0; (*Next State*)
				RETURN;

			ELSE
				SoftStop := TRUE;

			END_IF
		END_IF

		IF SoftStop THEN
			EVP_Out_Eng_Tgt := EVP_Out_Eng_Tgt - CFG.EVP_Out_Eng_Dec * CFG.Cycle;
			EVP_Out_Eng_Tgt := MIN(EVP_Out_Eng_Tgt, CFG.EVP_Out_Eng_Max);
			EVP_Out_Eng_Tgt := MIN(EVP_Out_Eng_Tgt, CFG.EVP_Out_Eng_Min - DeltaLS * CFG.EVP_Out_Eng_K);
			EVP_Out_Eng_Tgt := MAX(EVP_Out_Eng_Tgt, CFG.EVP_Out_Eng_Min);

			IF EVP_Out_Eng_Tgt = CFG.EVP_Out_Eng_Min OR CFG.EVP_Out_Eng_Dec <= 0
			THEN EVP_Eng_O := 0;
			ELSE EVP_Eng_O := REAL_TO_UINT(EVP_Out_Eng_Tgt);
			END_IF

		ELSE
			EVP_Out_Eng_Tgt := EVP_Out_Eng_Tgt + CFG.EVP_Out_Eng_Inc * CFG.Cycle;
			EVP_Out_Eng_Tgt := MIN(EVP_Out_Eng_Tgt, CFG.EVP_Out_Eng_Max);
			EVP_Out_Eng_Tgt := MIN(EVP_Out_Eng_Tgt, CFG.EVP_Out_Eng_Min - DeltaLS * CFG.EVP_Out_Eng_K);
			EVP_Out_Eng_Tgt := MAX(EVP_Out_Eng_Tgt, CFG.EVP_Out_Eng_Min);

			EVP_Eng_O := REAL_TO_UINT(EVP_Out_Eng_Tgt);

		END_IF

		IF EVP_Eng_O = 0 THEN
			OUT_LP   := 0;
			State    := 0; (*Next State*)

		ELSE
			EVP_Out_Fill_Tgt := EVP_Out_Eng_Tgt * CFG.EVP_Out_Fill_K + CFg.EVP_Out_Fill_Off;
			EVP_Out_Fill_Tgt := MIN(EVP_Out_Fill_Tgt, CFG.EVP_Out_Fill_Max);
			EVP_Out_Fill_Tgt := MAX(EVP_Out_Fill_Tgt, CFG.EVP_Out_Fill_Min);
	
			EV_Eng_EI := TRUE;
			EV_Eng_PO := TRUE;
			EV_PP_O   := FALSE;
		(*	EVP_Eng_O*)
			P_Fill    := CFG.EVP_Out_P_Fill; (*bar*)
			EVP_Fill  := REAL_TO_INT(EVP_Out_Fill_Tgt * 10.0); (*%*)
			OUT_LP    := 1;

		END_IF

	ELSE
		IF Event_I = INIT_CONTINUOUS
		OR Event_O = INIT_CONTINUOUS OR State = 2000 AND Event_O = END_CONTINUOUS
		OR Event_C = INIT_CONTINUOUS OR State = 2100 AND Event_C = END_CONTINUOUS
		OR Event_F = INIT_CONTINUOUS
		OR Event_T = INIT_CONTINUOUS OR State = 2200 AND Event_T = END_CONTINUOUS

		THEN
			OUT_LP   := 0;
			State    := 0; (*Next State*)

		ELSE
			EV_Eng_EI := FALSE;
			EV_Eng_PO := FALSE;
			EV_PP_O   := TRUE;
			EVP_Eng_O := 0; (*mA*)
			P_Fill    := 0; (*bar*)
			EVP_Fill  := 0; (*%*)
			OUT_LP    := 1;

		END_IF
	END_IF

(*Float IN - Easing OUT*)
3000:
	IF TimeOut OR LS_Err OR LS_Pos < CFG.TgtLS_In OR (LS_BOARD_S.Err OR LS_BOARD_S.Pos < CFG.Board_S_Min_Out) AND LS_Pos < CFG.TgtLS_Safe_In THEN
		Out_LP := 0;
		State  := 0;  (*Next State*)

	ELSE
		(*Activate SoftStop*)
		IF Event_F <> NONE
		OR Event_I = INIT_CONTINUOUS
		OR Event_C = INIT_CONTINUOUS
		OR Event_O = INIT_CONTINUOUS
		OR Event_T = INIT_CONTINUOUS
		THEN

			(*If already stoping, full stop*)
			IF SoftStop THEN
				OUT_LP    := 0;
				State     := 0; (*Next State*)
				RETURN;

			ELSE
				SoftStop := TRUE;

			END_IF
		END_IF

		IF SoftStop THEN
			EVP_Out_FE_Tgt := EVP_Out_FE_Tgt - CFG.EVP_Out_FE_Dec * CFG.Cycle;
			EVP_Out_FE_Tgt := MIN(EVP_Out_FE_Tgt, CFG.EVP_Out_FE_Max);
			EVP_Out_FE_Tgt := MAX(EVP_Out_FE_Tgt, CFG.EVP_Out_FE_Min);

			IF EVP_Out_FE_Tgt = CFG.EVP_Out_FE_Min THEN
				EVP_Out_SE_Tgt := EVP_Out_SE_Tgt - CFG.EVP_Out_SE_Dec * CFG.Cycle;
				EVP_Out_SE_Tgt := MIN(EVP_Out_SE_Tgt, CFG.EVP_Out_SE_Max);
				EVP_Out_SE_Tgt := MAX(EVP_Out_SE_Tgt, CFG.EVP_Out_SE_Min);
			END_IF

			IF EVP_Out_SE_Tgt = CFG.EVP_Out_SE_Min OR CFG.EVP_Out_SE_Dec <= 0
			THEN EVP_SE_O := 0;
			ELSE EVP_SE_O := REAL_TO_UINT(EVP_Out_SE_Tgt );
			END_IF

			IF EVP_Out_FE_Tgt = CFG.EVP_Out_FE_Min OR CFG.EVP_Out_FE_Dec <= 0
			THEN EVP_FE_O := 0;
			ELSE EVP_FE_O := REAL_TO_UINT(EVP_Out_FE_Tgt );
			END_IF

		ELSE
			EVP_Out_SE_Tgt := EVP_Out_SE_Tgt + CFG.EVP_Out_SE_Inc * CFG.Cycle;
			EVP_Out_SE_Tgt := MIN(EVP_Out_SE_Tgt, CFG.EVP_Out_SE_Max);
			EVP_Out_SE_Tgt := MAX(EVP_Out_SE_Tgt, CFG.EVP_Out_SE_Min);

			IF EVP_Out_SE_Tgt = CFG.EVP_Out_SE_Man OR EVP_Out_SE_Tgt = CFG.EVP_Out_SE_Max THEN
				EVP_Out_FE_Tgt := EVP_Out_FE_Tgt + CFG.EVP_Out_FE_Inc * CFG.Cycle;
				EVP_Out_FE_Tgt := MIN(EVP_Out_FE_Tgt, CFG.EVP_Out_FE_Max);
				EVP_Out_FE_Tgt := MAX(EVP_Out_FE_Tgt, CFG.EVP_Out_FE_Min);
			END_IF

			EVP_SE_O  := REAL_TO_UINT(EVP_Out_SE_Tgt);
			EVP_FE_O  := REAL_TO_UINT(EVP_Out_FE_Tgt);

		END_IF

		(*If ALL stopped go to Init State*)
		IF EVP_SE_O = 0 AND EVP_FE_O = 0 THEN
			Out_LP := 0;
			State  := 0;  (*Next State*)

		END_IF
	END_IF

(*Float OUT - Easing IN*)
4000:
	IF TimeOut OR LS_Err OR LS_Pos > CFG.TgtLS_Out OR (LS_BOARD_P.Err OR LS_BOARD_P.Pos < CFG.Board_P_Min_Out) AND LS_Pos > CFG.TgtLS_Safe_Out THEN
		Out_LP := 0;
		State  := 0;  (*Next State*)

	ELSE
		(*Activate SoftStop*)
		IF Event_F <> NONE
		OR Event_I = INIT_CONTINUOUS
		OR Event_C = INIT_CONTINUOUS
		OR Event_O = INIT_CONTINUOUS
		OR Event_T = INIT_CONTINUOUS
		THEN

			(*If already stoping, full stop*)
			IF SoftStop THEN
				OUT_LP    := 0;
				State     := 0; (*Next State*)
				RETURN;

			ELSE
				SoftStop := TRUE;

			END_IF
		END_IF

		IF SoftStop THEN
			EVP_In_FE_Tgt := EVP_In_FE_Tgt - CFG.EVP_In_FE_Dec * CFG.Cycle;
			EVP_In_FE_Tgt := MIN(EVP_In_FE_Tgt, CFG.EVP_In_FE_Max);
			EVP_In_FE_Tgt := MAX(EVP_In_FE_Tgt, CFG.EVP_In_FE_Min);

			IF EVP_In_FE_Tgt = CFG.EVP_In_FE_Min THEN
				EVP_In_SE_Tgt := EVP_In_SE_Tgt - CFG.EVP_In_SE_Dec * CFG.Cycle;
				EVP_In_SE_Tgt := MIN(EVP_In_SE_Tgt, CFG.EVP_In_SE_Max);
				EVP_In_SE_Tgt := MAX(EVP_In_SE_Tgt, CFG.EVP_In_SE_Min);
			END_IF

			IF EVP_In_SE_Tgt = CFG.EVP_In_SE_Min OR CFG.EVP_In_SE_Dec <= 0
			THEN EVP_SE_I := 0;
			ELSE EVP_SE_I := REAL_TO_UINT(EVP_In_SE_Tgt );
			END_IF

			IF EVP_In_FE_Tgt = CFG.EVP_In_FE_Min OR CFG.EVP_In_FE_Dec <= 0
			THEN EVP_FE_I := 0;
			ELSE EVP_FE_I := REAL_TO_UINT(EVP_In_FE_Tgt );
			END_IF

		ELSE
			EVP_In_SE_Tgt := EVP_In_SE_Tgt + CFG.EVP_In_SE_Inc * CFG.Cycle;
			EVP_In_SE_Tgt := MIN(EVP_In_SE_Tgt, CFG.EVP_In_SE_Max);
			EVP_In_SE_Tgt := MAX(EVP_In_SE_Tgt, CFG.EVP_In_SE_Min);
	
			IF EVP_In_SE_Tgt = CFG.EVP_In_SE_Man OR EVP_In_SE_Tgt = CFG.EVP_In_SE_Max THEN
				EVP_In_FE_Tgt := EVP_In_FE_Tgt + CFG.EVP_In_FE_Inc * CFG.Cycle;
				EVP_In_FE_Tgt := MIN(EVP_In_FE_Tgt, CFG.EVP_In_FE_Max);
				EVP_In_FE_Tgt := MAX(EVP_In_FE_Tgt, CFG.EVP_In_FE_Min);
			END_IF
	
			EVP_SE_I  := REAL_TO_UINT(EVP_In_SE_Tgt );
			EVP_FE_I  := REAL_TO_UINT(EVP_In_FE_Tgt );

		END_IF

		(*If ALL stopped go to Init State*)
		IF EVP_SE_I = 0 AND EVP_FE_I = 0 THEN
			Out_LP := 0;
			State  := 0;  (*Next State*)

		END_IF
	END_IF

END_CASE



(*hacer float antes de empezar a pompar cuando mueve de un lado al otro.*)
(*El float antes de mover tendra que ser en funcion de la velocidad, es decir delta de la posicion.*)
END_FUNCTION_BLOCK

(* POU FB/FB_TRAVELLER, ST *)
FUNCTION_BLOCK FB_TRAVELLER
VAR_INPUT
	Enable : BOOL;
	Ready  : BOOL;
	Perc   : REAL;

	IN_A : ARRAY[1..3] OF BOOL;
	IN_B : ARRAY[1..3] OF BOOL;
	IN_T : ARRAY[1..2] OF BOOL;
	IN_D : ARRAY[1..2] OF BOOL;
END_VAR
VAR_IN_OUT
	P_A : ST_SENSOR_BAR;
	P_B : ST_SENSOR_BAR;
	LS  : ST_SENSOR_POS;
	CFG : ST_TRAVELLER_CFG;
END_VAR
VAR_OUTPUT
	OUT_EVRA : BOOL;
	OUT_EVRB : BOOL;
	OUT_EVAB : BOOL;

	OUT_EVPA : BOOL;
	OUT_EVPB : BOOL;

	OUT_TWC : INT;
	OUT_LP  : BYTE;
	OUT_HP  : BYTE;
END_VAR
VAR
	State   : WORD;

	IN_Hmi_A : BOOL;
	IN_Hmi_B : BOOL;
	IN_Hmi_T : BOOL;
	IN_Hmi_D : BOOL;

	SIA  : ARRAY[1..4] OF FB_SMART_INPUT;
	SIB  : ARRAY[1..4] OF FB_SMART_INPUT;
	SIT  : ARRAY[1..3] OF FB_SMART_INPUT;
	SID  : ARRAY[1..3] OF FB_SMART_INPUT;

	EventA  : EN_SMART_INPUT_STATE;
	EventB  : EN_SMART_INPUT_STATE;
	EventT  : EN_SMART_INPUT_STATE;
	EventD  : EN_SMART_INPUT_STATE;

	Spd_Tgt  : REAL;
	SoftStop : BOOL;

	TimeCnt : REAL;
	TimeOut : BOOL;

	P_Bypass  : BOOL;

	Slow : BOOL;
	LS_Dif : REAL;
	LS_Tgt : REAL;

	LS_Min : BOOL;
	LS_Max : BOOL;
	LS_Mid : BOOL;
	P_Dw   : BOOL;

	Hyst_Cnt : REAL;
	Hyst_ON  : BOOL;

	Move_A : BOOL;
	Move_B : BOOL;

	ToFaroValue : REAL;

END_VAR
(*A->IN->Stbd*)

LS_Max := NOT LS.Err AND LS.Pos > CFG.TgtLS_Max  - CFG.LS_DB;
LS_Min := NOT LS.Err AND LS.Pos < CFG.TgtLS_Min  + CFG.LS_DB;
LS_Mid := NOT LS.Err AND LS.Pos < CFG.TgtLS_Zero + CFG.LS_DB AND LS.Pos > CFG.TgtLS_Zero - CFG.LS_DB;

(*Check Inputs*)
SIA[1](In:= IN_A[1],  T_Cont:= T#0ms, T_DClk:= T#0ms);
SIA[2](In:= IN_A[2],  T_Cont:= T#0ms, T_DClk:= T#0ms);
SIA[3](In:= IN_A[3],  T_Cont:= T#0ms, T_DClk:= T#0ms);
SIA[4](In:= IN_Hmi_A, T_Cont:= T#0ms, T_DClk:= T#0ms);

SIB[1](In:= IN_B[1],  T_Cont:= T#0ms, T_DClk:= T#0ms);
SIB[2](In:= IN_B[2],  T_Cont:= T#0ms, T_DClk:= T#0ms);
SIB[3](In:= IN_B[3],  T_Cont:= T#0ms, T_DClk:= T#0ms);
SIB[4](In:= IN_Hmi_B, T_Cont:= T#0ms, T_DClk:= T#0ms);

SIT[1](In:= IN_T[1],  T_Cont:= T#200ms, T_DClk:= T#0ms);
SIT[2](In:= IN_T[2],  T_Cont:= T#200ms, T_DClk:= T#0ms);
SIT[3](In:= IN_Hmi_T, T_Cont:= T#200ms, T_DClk:= T#0ms);

SID[1](In:= IN_D[1],  T_Cont:= T#0ms, T_DClk:= T#0ms);
SID[2](In:= IN_D[2],  T_Cont:= T#0ms, T_DClk:= T#0ms);
SID[3](In:= IN_Hmi_D, T_Cont:= T#0ms, T_DClk:= T#0ms);

IF NOT Enable THEN
	OUT_EVRA := FALSE;
	OUT_EVRB := FALSE;
	OUT_EVAB := FALSE;

	OUT_EVPA := FALSE;
	OUT_EVPB := FALSE;

	ToFaroValue := 0.0;

	OUT_TWC  := 0;
	OUT_LP   := 0;
	OUT_HP   := 0;

	TimeCnt  := 0.0;
	State    := 0;
	RETURN;
END_IF

(*Check Time*)
TimeOut := TimeOut OR ( CFG.TimeMax > 0  AND TimeCnt > CFG.TimeMax );
TimeCnt := TimeCnt + CFG.Cycle;

IF    SIA[1].Event <> NONE THEN EventA := SIA[1].Event;
ELSIF SIA[2].Event <> NONE THEN EventA := SIA[2].Event;
ELSIF SIA[3].Event <> NONE THEN EventA := SIA[3].Event;
ELSIF SIA[4].Event <> NONE THEN EventA := SIA[4].Event;
ELSE							EventA := NONE;
END_IF

IF    SIB[1].Event <> NONE THEN EventB := SIB[1].Event;
ELSIF SIB[2].Event <> NONE THEN EventB := SIB[2].Event;
ELSIF SIB[3].Event <> NONE THEN EventB := SIB[3].Event;
ELSIF SIB[4].Event <> NONE THEN EventB := SIB[4].Event;
ELSE							EventB := NONE;
END_IF

IF    SIT[1].Event <> NONE THEN EventT := SIT[1].Event;
ELSIF SIT[2].Event <> NONE THEN EventT := SIT[2].Event;
ELSIF SIT[3].Event <> NONE THEN EventT := SIT[3].Event;
ELSE							EventT := NONE;
END_IF

IF    SID[1].Event <> NONE THEN EventD := SID[1].Event;
ELSIF SID[2].Event <> NONE THEN EventD := SID[2].Event;
ELSIF SID[3].Event <> NONE THEN EventD := SID[3].Event;
ELSE							EventD := NONE;
END_IF

(*Working States*)
CASE State OF

(*Init State*)
0:
	OUT_EVRA := FALSE;
	OUT_EVRB := FALSE;
	OUT_EVAB := FALSE;
	OUT_TWC  := 0;
	OUT_LP   := 0;

	SoftStop := FALSE;
    TimeCnt  := 0.0; (*Time Count*)

	(*Start IN*)
	IF EventA = INIT_CONTINUOUS AND Ready THEN
		Spd_Tgt := CFG.MinEVPA;
		TimeOut := FALSE; (*Reset TimeOut Error*)
		State   := 100;   (*Next State*)

	(*Start OUT*)
	ELSIF EventB = INIT_CONTINUOUS AND Ready THEN
		Spd_Tgt := CFG.MinEVPB;
		TimeOut := FALSE; (*Reset TimeOut Error*)
		State   := 200;   (*Next State*)

	(*Start TACK*)
	ELSIF EventT = INIT_CONTINUOUS AND Ready THEN
		TimeOut := FALSE; (*Reset TimeOut Error*)
		State   := 300;   (*Next State*)

	(*Start DUMP*)
	ELSIF EventD = INIT_CONTINUOUS THEN
		TimeOut := FALSE; (*Reset TimeOut Error*)
		State   := 400;   (*Next State*)

	END_IF

(*Manual A-IN*)
100:
	IF EventD = INIT_CONTINUOUS THEN
		OUT_EVRA := FALSE;
		OUT_EVRB := FALSE;
		OUT_EVAB := TRUE;
		OUT_TWC  := 0;
		OUT_LP   := 0;

		TimeCnt  := 0.0; (*Time Count*)
		State    := 400; (*Next State*)

	ELSIF NOT Ready OR TimeOut OR P_A.AlMax THEN
		OUT_TWC := 0;
		OUT_LP  := 0;
		State   := 0;  (*Next State*)

	ELSIF EventB = INIT_CONTINUOUS THEN
		OUT_EVRA := FALSE;
		OUT_EVRB := FALSE;
		OUT_EVAB := FALSE;
		OUT_TWC  := 0;
		OUT_LP   := 0;

		Spd_Tgt  := CFG.MinEVPB;
		TimeCnt  := 0.0; (*Time Count*)
		State    := 200; (*Next State*)

	ELSIF CFG.LS_Limit AND LS.Pos < CFG.TgtLS_Min + CFG.LS_DB THEN
		OUT_EVRB := FALSE;
		OUT_TWC  := 0;
		OUT_LP   := 0;
		State    := 0;  (*Next State*)

	ELSE
		IF EventA = END_CONTINUOUS THEN
			(*If already stoping, full stop*)
			IF SoftStop THEN
				OUT_TWC := 0;
				OUT_LP  := 0;
				State   := 0; (*Next State*)
				RETURN;

			ELSE
				SoftStop := TRUE;

			END_IF
		END_IF

		LS_Dif := ABS(LS.Pos - CFG.TgtLS_Min);

		IF SoftStop THEN
			Spd_Tgt  := Spd_Tgt - CFG.Spd_Dec * CFG.Cycle;

			IF CFG.LS_Limit AND LS_Dif < CFG.LS_Dist THEN (*Si Dist = 0 nunca entrara*)
				Spd_Tgt := MIN(Spd_Tgt, CFG.MinEVPA + LS_Dif * ((CFG.MaxEVPA - CFG.MinEVPA) / CFG.LS_Dist));
			END_IF

			Spd_Tgt  := MIN(Spd_Tgt, CFG.MaxEVPA);
			Spd_Tgt  := MAX(Spd_Tgt, CFG.MinEVPA);

			IF Spd_Tgt = CFG.MinEVPA OR CFG.Spd_Dec <= 0 THEN
				OUT_EVRB := FALSE;
				OUT_TWC  := 0;
				OUT_LP   := 0;
				State    := 0; (*Next State*);

			ELSE
				OUT_EVRB := TRUE;
				OUT_TWC  := REAL_TO_INT(Spd_Tgt * Perc * 10.0);
				OUT_LP   := 1;
				Slow     := TRUE;
			END_IF

		ELSE
			Spd_Tgt  := Spd_Tgt + CFG.Spd_Inc * CFG.Cycle;

			IF CFG.LS_Limit AND LS_Dif < CFG.LS_Dist THEN (*Si Dist = 0 nunca entrara*)
				Spd_Tgt := MIN(Spd_Tgt, CFG.MinEVPA + LS_Dif * ((CFG.MaxEVPA - CFG.MinEVPA) / CFG.LS_Dist));
				OUT_LP  := 1;
				Slow    := TRUE;
			ELSE
				OUT_LP  := CFG.LP;
				Slow    := FALSE;
			END_IF

			Spd_Tgt  := MIN(Spd_Tgt, CFG.MaxEVPA);
			Spd_Tgt  := MAX(Spd_Tgt, CFG.MinEVPA);

			OUT_EVRB := TRUE;
			OUT_TWC  := REAL_TO_INT(Spd_Tgt * Perc * 10.0);

		END_IF

	END_IF

(*Manual B-OUT*)
200:
	IF EventD = INIT_CONTINUOUS THEN
		OUT_EVRA := FALSE;
		OUT_EVRB := FALSE;
		OUT_EVAB := TRUE;
		OUT_TWC  := 0;
		OUT_LP   := 0;

		TimeCnt  := 0.0; (*Time Count*)
		State    := 400; (*Next State*)

	ELSIF NOT Ready OR TimeOut OR P_B.AlMax THEN
		OUT_TWC := 0;
		OUT_LP  := 0;
		State   := 0;  (*Next State*)

	ELSIF EventA = INIT_CONTINUOUS THEN
		OUT_EVRA := FALSE;
		OUT_EVRB := FALSE;
		OUT_EVAB := FALSE;
		OUT_TWC  := 0;
		OUT_LP   := 0;

		Spd_Tgt := CFG.MinEVPA;
		TimeCnt  := 0.0; (*Time Count*)
		State    := 100;   (*Next State*)

	ELSIF CFG.LS_Limit AND LS.Pos > CFG.TgtLS_Max - CFG.LS_DB THEN
		OUT_EVRA := FALSE;
		OUT_TWC  := 0;
		OUT_LP   := 0;
		State    := 0;  (*Next State*)

	ELSE
		IF EventB = END_CONTINUOUS THEN
			(*If already stoping, full stop*)
			IF SoftStop THEN
				OUT_TWC := 0;
				OUT_LP  := 0;
				State   := 0; (*Next State*)
				RETURN;

			ELSE
				SoftStop := TRUE;

			END_IF
		END_IF

		LS_Dif := ABS(LS.Pos - CFG.TgtLS_Min);

		IF SoftStop THEN
			Spd_Tgt  := Spd_Tgt - CFG.Spd_Dec * CFG.Cycle;

			IF CFG.LS_Limit AND LS_Dif < CFG.LS_Dist THEN (*Si Dist = 0 nunca entrara*)
				Spd_Tgt := MIN(Spd_Tgt, CFG.MinEVPB + LS_Dif * ((CFG.MaxEVPB - CFG.MinEVPB) / CFG.LS_Dist));
			END_IF

			Spd_Tgt  := MIN(Spd_Tgt, CFG.MaxEVPB);
			Spd_Tgt  := MAX(Spd_Tgt, CFG.MinEVPB);

			IF Spd_Tgt = CFG.MinEVPB OR CFG.Spd_Dec <= 0 THEN
				OUT_EVRA := FALSE;
				OUT_TWC  := 0;
				OUT_LP   := 0;
				State    := 0; (*Next State*);

			ELSE
				OUT_EVRA := TRUE;
				OUT_TWC  := REAL_TO_INT(-Spd_Tgt * Perc * 10.0);
				OUT_LP   := 1;
				Slow     := TRUE;
			END_IF

		ELSE
			Spd_Tgt  := Spd_Tgt + CFG.Spd_Inc * CFG.Cycle;

			IF CFG.LS_Limit AND LS_Dif < CFG.LS_Dist THEN (*Si Dist = 0 nunca entrara*)
				Spd_Tgt := MIN(Spd_Tgt, CFG.MinEVPB + LS_Dif * ((CFG.MaxEVPB - CFG.MinEVPB) / CFG.LS_Dist));
				OUT_LP  := 1;
				Slow    := TRUE;
			ELSE
				OUT_LP  := CFG.LP;
				Slow    := FALSE;
			END_IF

			Spd_Tgt  := MIN(Spd_Tgt, CFG.MaxEVPB);
			Spd_Tgt  := MAX(Spd_Tgt, CFG.MinEVPB);

			OUT_EVRA := TRUE;
			OUT_TWC  := REAL_TO_INT(-Spd_Tgt * Perc * 10.0);

		END_IF

	END_IF

(*Init TACK*)
300:
	IF EventD = INIT_CONTINUOUS THEN
		OUT_EVAB := TRUE;

		State    := 400; (*Next State*)

	ELSIF EventT = INIT_CONTINUOUS OR NOT Ready OR TimeOut OR P_A.AlMax OR P_B.AlMax OR LS.Err THEN
		State    := 0;   (*Next State*)

	ELSIF EventA = INIT_CONTINUOUS THEN
		Spd_Tgt  := CFG.MinEVPA;
		State    := 100; (*Next State*)

	ELSIF EventB = INIT_CONTINUOUS THEN
		Spd_Tgt  := CFG.MinEVPB;
		State    := 200; (*Next State*)

	ELSIF LS.Pos + CFG.TgtLS_Tack_Off > CFG.TgtLS_Zero THEN
		LS_Tgt   := CFG.TgtLS_Zero + CFG.TgtLS_Zero - LS.Pos - CFG.TgtLS_Tack_Off;

		IF CFG.LS_Limit THEN LS_Tgt := MAX(LS_Tgt, CFG.TgtLS_Min); END_IF

		Spd_Tgt  := CFG.MinEVPA;
		State    := 500; (*Next State*)

	ELSIF LS.Pos - CFG.TgtLS_Tack_Off < CFG.TgtLS_Zero THEN
		LS_Tgt   := CFG.TgtLS_Zero + CFG.TgtLS_Zero - LS.Pos + CFG.TgtLS_Tack_Off;

		IF CFG.LS_Limit THEN LS_Tgt := MIN(LS_Tgt, CFG.TgtLS_Max); END_IF

		Spd_Tgt  := CFG.MinEVPB;
		State    := 600; (*Next State*)

	ELSE
		State    := 0;   (*Next State*)

	END_IF

(*DUMP*)
400:
	IF EventD = END_CONTINUOUS OR TimeOut THEN
		OUT_EVAB := FALSE;
		State    := 0;  (*Next State*)

	ELSIF CFG.LS_Limit AND ( LS.Pos >= CFG.TgtLS_Max OR LS.Pos <= CFG.TgtLS_Min ) THEN
		OUT_EVAB := FALSE;
		State    := 0;  (*Next State*)

	ELSE
		OUT_EVAB := TRUE;

	END_IF

(*Init Auto IN*)
500:
	IF EventD = INIT_CONTINUOUS THEN
		OUT_EVRA := FALSE;
		OUT_EVRB := FALSE;
		OUT_EVAB := TRUE;
		OUT_TWC  := 0;
		OUT_LP   := 0;

		TimeCnt  := 0.0; (*Time Count*)
		State    := 400;   (*Next State*)

	ELSIF NOT Ready OR TimeOut OR P_A.AlMax OR LS.Err THEN
		OUT_TWC  := 0;
		OUT_LP   := 0;
		State    := 0;  (*Next State*)

	ELSIF EventA = INIT_CONTINUOUS THEN
		OUT_EVRA := FALSE;
		OUT_EVRB := FALSE;
		OUT_EVAB := FALSE;
		OUT_TWC  := 0;
		OUT_LP   := 0;

		Spd_Tgt  := CFG.MinEVPA;
		TimeCnt  := 0.0; (*Time Count*)
		State    := 100; (*Next State*)

	ELSIF EventB = INIT_CONTINUOUS THEN
		OUT_EVRA := FALSE;
		OUT_EVRB := FALSE;
		OUT_EVAB := FALSE;
		OUT_TWC  := 0;
		OUT_LP   := 0;

		Spd_Tgt  := CFG.MinEVPB;
		TimeCnt  := 0.0; (*Time Count*)
		State    := 200; (*Next State*)

	ELSIF LS.Pos < LS_Tgt + CFG.LS_DB THEN
		OUT_EVRB := FALSE;
		OUT_TWC  := 0;
		OUT_LP   := 0;
		State    := 0;   (*Next State*)

	ELSE
		IF EventT = INIT_CONTINUOUS THEN
			(*If already stoping, full stop*)
			IF SoftStop THEN
				OUT_TWC := 0;
				OUT_LP  := 0;
				State   := 0; (*Next State*)
				RETURN;

			ELSE
				SoftStop := TRUE;

			END_IF
		END_IF

		LS_Dif := ABS(LS.Pos - LS_Tgt);

		IF SoftStop THEN
			Spd_Tgt  := Spd_Tgt - CFG.Spd_Dec * CFG.Cycle;

			IF LS_Dif < CFG.LS_Dist THEN (*Si Dist = 0 nunca entrara*)
				Spd_Tgt := MIN(Spd_Tgt, CFG.MinEVPA + LS_Dif * ((CFG.MaxEVPA - CFG.MinEVPA) / CFG.LS_Dist));
			END_IF

			Spd_Tgt  := MIN(Spd_Tgt, CFG.MaxEVPA);
			Spd_Tgt  := MAX(Spd_Tgt, CFG.MinEVPA);

			IF Spd_Tgt = CFG.MinEVPA OR CFG.Spd_Dec <= 0 THEN
				OUT_EVRB := FALSE;
				OUT_TWC  := 0;
				OUT_LP   := 0;
				State    := 0; (*Next State*);

			ELSE
				OUT_EVRB := TRUE;
				OUT_TWC  := REAL_TO_INT(Spd_Tgt * Perc * 10.0);
				OUT_LP   := 1;
				Slow     := TRUE;
			END_IF

		ELSE
			Spd_Tgt  := Spd_Tgt + CFG.Spd_Inc * CFG.Cycle;

			IF LS_Dif < CFG.LS_Dist THEN (*Si Dist = 0 nunca entrara*)
				Spd_Tgt := MIN(Spd_Tgt, CFG.MinEVPA + LS_Dif * ((CFG.MaxEVPA - CFG.MinEVPA) / CFG.LS_Dist));
				OUT_LP  := 1;
				Slow    := TRUE;
			ELSE
				OUT_LP  := CFG.LP;
				Slow    := FALSE;
			END_IF

			Spd_Tgt  := MIN(Spd_Tgt, CFG.MaxEVPA);
			Spd_Tgt  := MAX(Spd_Tgt, CFG.MinEVPA);

			OUT_EVRB := TRUE;
			OUT_TWC  := REAL_TO_INT(Spd_Tgt * Perc * 10.0);

		END_IF

	END_IF

(*Init Auto OUT*)
600:
	IF EventD = INIT_CONTINUOUS THEN
		OUT_EVRA := FALSE;
		OUT_EVRB := FALSE;
		OUT_EVAB := TRUE;
		OUT_TWC  := 0;
		OUT_LP   := 0;

		TimeCnt  := 0.0; (*Time Count*)
		State    := 400; (*Next State*)

	ELSIF NOT Ready OR TimeOut OR P_B.AlMax OR LS.Err THEN
		OUT_TWC  := 0;
		OUT_LP   := 0;
		State    := 0;  (*Next State*)

	ELSIF EventA = INIT_CONTINUOUS THEN
		OUT_EVRA := FALSE;
		OUT_EVRB := FALSE;
		OUT_EVAB := FALSE;
		OUT_TWC  := 0;
		OUT_LP   := 0;

		Spd_Tgt  := CFG.MinEVPA;
		TimeCnt  := 0.0; (*Time Count*)
		State    := 100; (*Next State*)

	ELSIF EventB = INIT_CONTINUOUS THEN
		OUT_EVRA := FALSE;
		OUT_EVRB := FALSE;
		OUT_EVAB := FALSE;
		OUT_TWC  := 0;
		OUT_LP   := 0;

		Spd_Tgt  := CFG.MinEVPB;
		TimeCnt  := 0.0; (*Time Count*)
		State    := 200;   (*Next State*)

	ELSIF LS.Pos > LS_Tgt - CFG.LS_DB THEN
		OUT_EVRA := FALSE;
		OUT_TWC  := 0;
		OUT_LP   := 0;
		State    := 0;  (*Next State*)

	ELSE
		IF EventT = INIT_CONTINUOUS THEN
			(*If already stoping, full stop*)
			IF SoftStop THEN
				OUT_TWC := 0;
				OUT_LP  := 0;
				State   := 0; (*Next State*)
				RETURN;

			ELSE
				SoftStop := TRUE;

			END_IF
		END_IF

		LS_Dif := ABS(LS.Pos - LS_Tgt);

		IF SoftStop THEN
			Spd_Tgt  := Spd_Tgt - CFG.Spd_Dec * CFG.Cycle;

			IF CFG.LS_Limit AND LS_Dif < CFG.LS_Dist THEN (*Si Dist = 0 nunca entrara*)
				Spd_Tgt := MIN(Spd_Tgt, CFG.MinEVPB + LS_Dif * ((CFG.MaxEVPB - CFG.MinEVPB) / CFG.LS_Dist));
			END_IF

			Spd_Tgt  := MIN(Spd_Tgt, CFG.MaxEVPB);
			Spd_Tgt  := MAX(Spd_Tgt, CFG.MinEVPB);

			IF Spd_Tgt = CFG.MinEVPB OR CFG.Spd_Dec <= 0 THEN
				OUT_EVRA := FALSE;
				OUT_TWC  := 0;
				OUT_LP   := 0;
				State    := 0; (*Next State*);

			ELSE
				OUT_EVRA := TRUE;
				OUT_TWC  := REAL_TO_INT(-Spd_Tgt * Perc * 10.0);
				OUT_LP   := 1;
				Slow     := TRUE;
			END_IF

		ELSE
			Spd_Tgt  := Spd_Tgt + CFG.Spd_Inc * CFG.Cycle;

			IF CFG.LS_Limit AND LS_Dif < CFG.LS_Dist THEN (*Si Dist = 0 nunca entrara*)
				Spd_Tgt := MIN(Spd_Tgt, CFG.MinEVPB + LS_Dif * ((CFG.MaxEVPB - CFG.MinEVPB) / CFG.LS_Dist));
				OUT_LP  := 1;
				Slow    := TRUE;
			ELSE
				OUT_LP  := CFG.LP;
				Slow    := FALSE;
			END_IF

			Spd_Tgt  := MIN(Spd_Tgt, CFG.MaxEVPB);
			Spd_Tgt  := MAX(Spd_Tgt, CFG.MinEVPB);

			OUT_EVRA := TRUE;
			OUT_TWC  := REAL_TO_INT(-Spd_Tgt * Perc * 10.0);

		END_IF

	END_IF

END_CASE

(*Evaluo HP*)
IF Hyst_Cnt > CFG.Hyst_TM THEN
	Hyst_ON := TRUE;
ELSE
	Hyst_ON  := FALSE;
	Hyst_Cnt := Hyst_Cnt + CFG.Cycle;
END_IF

IF OUT_TWC > 0 THEN
	IF P_A.Bar > CFG.Hyst_HP AND Hyst_ON OR P_A.Err THEN
		OUT_EVPA := TRUE;
		OUT_EVPB := FALSE;
		OUT_HP   := CFG.HP;
		Hyst_cnt := 0.0;

		ToFaroValue := 1.0;

	ELSIF P_A.Bar < CFG.Hyst_LP AND Hyst_ON THEN
		OUT_EVPA := FALSE;
		OUT_EVPB := FALSE;
		OUT_HP   := 0;
		Hyst_cnt := 0.0;

		ToFaroValue := 0.0;

	END_IF

	IF OUT_EVPA THEN
		OUT_EVRA := FALSE;
		OUT_EVRB := FALSE;
		OUT_TWC  := 0;
		OUT_LP   := 0;
	END_IF

ELSIF OUT_TWC < 0 THEN
	IF P_B.Bar > CFG.Hyst_HP AND Hyst_ON OR P_B.Err THEN
		OUT_EVPA := FALSE;
		OUT_EVPB := TRUE;
		OUT_HP   := CFG.HP;
		Hyst_cnt := 0.0;

		ToFaroValue := -1.0;

	ELSIF P_B.Bar < CFG.Hyst_LP AND Hyst_ON THEN
		OUT_EVPA := FALSE;
		OUT_EVPB := FALSE;
		OUT_HP   := 0;
		Hyst_cnt := 0.0;

		ToFaroValue := 0.0;

	END_IF

	IF OUT_EVPB THEN
		OUT_EVRA := FALSE;
		OUT_EVRB := FALSE;
		OUT_TWC  := 0;
		OUT_LP   := 0;
	END_IF

ELSE
	OUT_EVPA := FALSE;
	OUT_EVPB := FALSE;
	OUT_HP   := 0;

END_IF

Move_A := OUT_EVRB OR OUT_EVPA;
Move_B := OUT_EVRA OR OUT_EVPB;
END_FUNCTION_BLOCK

(* POU FB/FB_LP_FUNC_SF, ST *)
FUNCTION_BLOCK FB_LP_FUNC_SF
VAR_INPUT
	Enable : BOOL;
	Ready  : BOOL;

	Perc : REAL;

	IN_1   : BOOL;
	IN_2   : BOOL;

	IN_SF1 : BOOL;
	IN_SF2 : BOOL;

END_VAR
VAR_IN_OUT
	CFG : ST_LP_FUNC_CFG;
END_VAR
VAR_OUTPUT
	OUT_TWC : INT;
	OUT_LP  : BYTE;
END_VAR
VAR
	State : WORD;

	IN_Hmi_1 : BOOL;
	IN_Hmi_2 : BOOL;
	IN_SFA   : BOOL;
	IN_SFB   : BOOL;

	SI_A : FB_SMART_INPUT;
	SI_B : FB_SMART_INPUT;
	SI_Hmi_A : FB_SMART_INPUT;
	SI_Hmi_B : FB_SMART_INPUT;

	Spd_Tgt  : REAL;
	SoftStop : BOOL;

	CyclCnt : REAL;
	TimeOut : BOOL;

	SpdA : INT;
	SpdB : INT;
	Out_1: BOOL;
	Out_2: BOOL;
END_VAR
IF Cfg.A_Spd1 THEN
	SpdA := 1;
	SpdB := 2;

	SI_A(In:= IN_1, T_Cont:= T#0ms, T_DClk:= T#0ms);
	SI_B(In:= IN_2, T_Cont:= T#0ms, T_DClk:= T#0ms);

	SI_Hmi_A(In:= IN_Hmi_1, T_Cont:= T#0ms, T_DClk:= T#0ms);
	SI_Hmi_B(In:= IN_Hmi_2, T_Cont:= T#0ms, T_DClk:= T#0ms);

	IN_SFA := IN_SF1 AND Cfg.SF1_Limit;
	IN_SFB := IN_SF2 AND Cfg.SF2_Limit;
ELSE
	SpdA := 2;
	SpdB := 1;

	SI_A(In:= IN_2, T_Cont:= T#0ms, T_DClk:= T#0ms);
	SI_B(In:= IN_1, T_Cont:= T#0ms, T_DClk:= T#0ms);

	SI_Hmi_A(In:= IN_Hmi_2, T_Cont:= T#0ms, T_DClk:= T#0ms);
	SI_Hmi_B(In:= IN_Hmi_1, T_Cont:= T#0ms, T_DClk:= T#0ms);

	IN_SFA := IN_SF2 AND Cfg.SF2_Limit;
	IN_SFB := IN_SF1 AND Cfg.SF1_Limit;
END_IF

IF NOT Enable THEN
	OUT_TWC := 0;
	OUT_LP  := 0;

	CyclCnt := 0;
	State   := 0;
	RETURN;
END_IF

(*Check Time*)
TimeOut := TimeOut OR (CFG.TimeMax > 0 AND CyclCnt > CFG.TimeMax);
CyclCnt := CyclCnt + CFG.Cycle;

CASE State OF
0: (*INIT*)
	OUT_TWC := 0;
	CyclCnt := 0;

	SoftStop := FALSE;

	IF Ready THEN
		IF (SI_A.Event = INIT_CONTINUOUS OR SI_Hmi_A.Event = INIT_CONTINUOUS) THEN
			Spd_Tgt := CFG.SpdA_Min;
			OUT_TWC := REAL_TO_INT(Spd_Tgt * Perc * 10.0);
			TimeOut := FALSE;
			State   := 10;

		ELSIF (SI_B.Event = INIT_CONTINUOUS OR SI_Hmi_B.Event = INIT_CONTINUOUS) THEN
			Spd_Tgt := CFG.SpdB_Min;
			OUT_TWC := REAL_TO_INT(-Spd_Tgt * Perc * 10.0);
			TimeOut := FALSE;
			State   := 20;

		END_IF
	END_IF

10: (*A*)
	IF TimeOut OR IN_SFA THEN
		OUT_TWC := 0;
		State   := 0;

	(*ELSIF SI_B.Event = INIT_CONTINUOUS OR SI_Hmi_B.Event = INIT_CONTINUOUS THEN
		Spd_Tgt := CFG.SpdB_Min;
		OUT_TWC := REAL_TO_INT(-Spd_Tgt * Perc * 10.0);
		TimeOut := FALSE;
		State   := 20;*)

	ELSE
		IF SI_A.Event = END_CONTINUOUS  OR SI_Hmi_A.Event = END_CONTINUOUS
		OR SI_B.Event = INIT_CONTINUOUS OR SI_Hmi_B.Event = INIT_CONTINUOUS
		THEN
			IF SoftStop THEN
				OUT_TWC  := 0;
				OUT_LP   := 0;
				State    := 0;
				RETURN;
			ELSE
				SoftStop := TRUE;
			END_IF
		END_IF

		IF SoftStop THEN
			Spd_Tgt := Spd_Tgt - CFG.Spd_Dec * CFG.Cycle;
			Spd_Tgt := MIN(Spd_Tgt, CFG.SpdA_Max);
			Spd_Tgt := MAX(Spd_Tgt, CFG.SpdA_Min);

			IF Spd_Tgt = CFG.SpdA_Min OR CFG.Spd_Dec <= 0
			THEN OUT_TWC := 0;
			ELSE OUT_TWC := REAL_TO_INT(Spd_Tgt * Perc * 10.0);
			END_IF

		ELSE
			Spd_Tgt := Spd_Tgt + CFG.Spd_Inc * CFG.Cycle;
			Spd_Tgt := MIN(Spd_Tgt, CFG.SpdA_Max);
			Spd_Tgt := MAX(Spd_Tgt, CFG.SpdA_Min);

			OUT_TWC := REAL_TO_INT(Spd_Tgt * Perc * 10.0);

		END_IF

		IF OUT_TWC = 0 THEN
			State    := 0; (*Next State*)
		END_IF

		(*OUT_TWC := REAL_TO_INT(CFG.SpdA * Perc * 10.0);*)

	END_IF

20: (*B*)
	IF TimeOut OR IN_SFB THEN
		OUT_TWC := 0;
		State   := 0;

	(*ELSIF SI_A.Event = INIT_CONTINUOUS OR SI_Hmi_A.Event = INIT_CONTINUOUS THEN
		Spd_Tgt := CFG.SpdA_Min;
		OUT_TWC := REAL_TO_INT(Spd_Tgt * Perc * 10.0);
		TimeOut := FALSE;
		State   := 10;*)

	ELSE
		IF SI_B.Event = END_CONTINUOUS  OR SI_Hmi_B.Event = END_CONTINUOUS
		OR SI_A.Event = INIT_CONTINUOUS OR SI_Hmi_A.Event = INIT_CONTINUOUS
		THEN
			IF SoftStop THEN
				OUT_TWC  := 0;
				OUT_LP   := 0;
				State    := 0;
				RETURN;
			ELSE
				SoftStop := TRUE;
			END_IF
		END_IF

		IF SoftStop THEN
			Spd_Tgt := Spd_Tgt - CFG.Spd_Dec * CFG.Cycle;
			Spd_Tgt := MIN(Spd_Tgt, CFG.SpdB_Max);
			Spd_Tgt := MAX(Spd_Tgt, CFG.SpdB_Min);

			IF Spd_Tgt = CFG.SpdB_Min OR CFG.Spd_Dec <= 0
			THEN OUT_TWC := 0;
			ELSE OUT_TWC := REAL_TO_INT(-Spd_Tgt * Perc * 10.0);
			END_IF

		ELSE
			Spd_Tgt := Spd_Tgt + CFG.Spd_Inc * CFG.Cycle;
			Spd_Tgt := MIN(Spd_Tgt, CFG.SpdB_Max);
			Spd_Tgt := MAX(Spd_Tgt, CFG.SpdB_Min);

			OUT_TWC := REAL_TO_INT(-Spd_Tgt * Perc * 10.0);

		END_IF

		IF OUT_TWC = 0 THEN
			State    := 0; (*Next State*)
		END_IF

		(*OUT_TWC := REAL_TO_INT(-CFG.SpdB * Perc * 10.0);*)

	END_IF

END_CASE

IF Cfg.A_Spd1 THEN
	Out_1 := OUT_TWC > 0;
	Out_2 := OUT_TWC < 0;
ELSE
	Out_1 := OUT_TWC < 0;
	Out_2 := OUT_TWC > 0;
END_IF

IF OUT_TWC = 0 THEN
	OUT_LP := 0;
ELSE
	OUT_LP := 1; (*How Many*)
END_IF
END_FUNCTION_BLOCK

(* POU FB/FB_TACK_VALVE, ST *)
FUNCTION_BLOCK FB_TACK_VALVE
VAR_INPUT
	Enable : BOOL;
	Manual : BOOL;
	Clear  : BOOL;

	Heel_Ready  : BOOL;
	Heel_Value  : REAL;

	Port_Ready : BOOL;
	Port_Open  : BOOL;
	Port_Close : BOOL;

	Stbd_Ready : BOOL;
	Stbd_Open  : BOOL;
	Stbd_Close : BOOL;

END_VAR
VAR_IN_OUT
	CFG : ST_TACK_VALVE_CFG;
END_VAR
VAR_OUTPUT
	OUT_Port_Open  : BOOL;
	OUT_Port_Close : BOOL;
	OUT_Stbd_Open  : BOOL;
	OUT_Stbd_Close : BOOL;
END_VAR
VAR
	State   : WORD;

	IN_Hmi_Port_Open  : BOOL;
	IN_Hmi_Port_Close : BOOL;
	IN_Hmi_Stbd_Open  : BOOL;
	IN_Hmi_Stbd_Close : BOOL;

	SI_Hmi_Port_Open  : FB_SMART_INPUT;
	SI_Hmi_Port_Close : FB_SMART_INPUT;
	SI_Hmi_Stbd_Open  : FB_SMART_INPUT;
	SI_Hmi_Stbd_Close : FB_SMART_INPUT;

	TimeCnt : REAL;
	TimeOut : BOOL;

	Alarm : ST_Alarm;

	Hyst_Cnt : REAL;
	Hyst_Old : WORD;

	StopEngine : BOOL;

END_VAR
IF Clear THEN
	Alarm.Alarm := FALSE;
	Alarm.Adver := FALSE;
	Alarm.AlCnt := 0;
	Alarm.AlLen := 0.0;
END_IF

(*Check Inputs*)
SI_Hmi_Port_Open (In:= IN_Hmi_Port_Open , T_Cont:= T#0ms, T_DClk:= T#0ms);
SI_Hmi_Port_Close(In:= IN_Hmi_Port_Close, T_Cont:= T#0ms, T_DClk:= T#0ms);
SI_Hmi_Stbd_Open (In:= IN_Hmi_Stbd_Open , T_Cont:= T#0ms, T_DClk:= T#0ms);
SI_Hmi_Stbd_Close(In:= IN_Hmi_Stbd_Close, T_Cont:= T#0ms, T_DClk:= T#0ms);

StopEngine := FALSE;

IF NOT Enable THEN
	OUT_Port_Open  := FALSE;
	OUT_Port_Close := FALSE;
	OUT_Stbd_Open  := FALSE;
	OUT_Stbd_Close := FALSE;

	Alarm.Alarm := FALSE;
	Alarm.Adver := FALSE;
	Alarm.AlCnt := 0;
	Alarm.AlLen := 0.0;

	TimeCnt := 0.0;
	State   := 0;
	RETURN;
END_IF

(*Check Time*)
TimeOut := TimeOut OR ( CFG.TimeMax > 0  AND TimeCnt > CFG.TimeMax );
TimeCnt := TimeCnt + CFG.Cycle;

(*Alarms*)
	IF NOT (Stbd_Open AND NOT Stbd_Close) AND NOT (Port_Open AND NOT Port_Close) THEN
		IF NOT Alarm.Alarm THEN
			Alarm.AlCnt  := Alarm.AlCnt + 1;
			Alarm.AlLen  := 0.0;
			Alarm.TimeInit := INPUTS.sLocal;
			Alarm.AlInit   := TRUE;

		ELSE
			Alarm.AlLen  := Alarm.AlLen + MAIN.Cycle_Time;

		END_IF

		Alarm.Adver := TRUE;
		Alarm.Alarm := TRUE;
		Alarm.Text  := '(TACK VALVE) Valve Not Open.';

		StopEngine := TRUE;

	ELSIF NOT Port_Ready OR NOT Stbd_Ready THEN
		IF NOT Alarm.Alarm THEN
			Alarm.AlCnt  := Alarm.AlCnt + 1;
			Alarm.AlLen  := 0.0;
			Alarm.TimeInit := INPUTS.sLocal;
			Alarm.AlInit   := TRUE;

		ELSE
			Alarm.AlLen  := Alarm.AlLen + MAIN.Cycle_Time;

		END_IF

		Alarm.Adver := TRUE;
		Alarm.Alarm := TRUE;

		Alarm.Text  := '(TACK VALVE) Valves Not Available.';

	ELSIF NOT Heel_Ready THEN
		IF NOT Alarm.Alarm THEN
			Alarm.AlCnt  := Alarm.AlCnt + 1;
			Alarm.AlLen  := 0.0;
			Alarm.TimeInit := INPUTS.sLocal;
			Alarm.AlInit   := TRUE;

		ELSE
			Alarm.AlLen  := Alarm.AlLen + MAIN.Cycle_Time;

		END_IF

		Alarm.Adver := TRUE;
		Alarm.Alarm := TRUE;

		Alarm.Text  := '(TACK VALVE) Heel Not Available.';

	ELSIF TimeOut THEN
		IF NOT Alarm.Alarm THEN
			Alarm.AlCnt  := Alarm.AlCnt + 1;
			Alarm.AlLen  := 0.0;
			Alarm.TimeInit := INPUTS.sLocal;
			Alarm.AlInit   := TRUE;

		ELSE
			Alarm.AlLen  := Alarm.AlLen + MAIN.Cycle_Time;

		END_IF

		Alarm.Adver := TRUE;
		Alarm.Alarm := TRUE;

		Alarm.Text  := '(TACK VALVE) TimeOut.';

	ELSE
		IF Alarm.Alarm THEN
			Alarm.TimeEnd := INPUTS.sLocal;
			Alarm.AlEnd   := TRUE;

		END_IF

			Alarm.Alarm := FALSE;

	END_IF

(*Working States*)
CASE State OF

(*Init State*)
0:
	OUT_Port_Open  := FALSE;
	OUT_Port_Close := FALSE;
	OUT_Stbd_Open  := FALSE;
	OUT_Stbd_Close := FALSE;

	TimeCnt := 0.0;

	(*Start Manual*)
	IF Manual THEN
		IF SI_Hmi_Port_Open.Event = INIT_CONTINUOUS THEN
			OUT_Port_Open := TRUE;

			TimeOut := FALSE; (*Reset TimeOut Error*)
			State   := 1001;  (*Next State*)

		ELSIF SI_Hmi_Port_Close.Event = INIT_CONTINUOUS THEN
			OUT_Port_Close := TRUE;

			TimeOut := FALSE; (*Reset TimeOut Error*)
			State   := 1002;  (*Next State*)

		ELSIF SI_Hmi_Stbd_Open.Event = INIT_CONTINUOUS THEN
			OUT_Stbd_Open := TRUE;

			TimeOut := FALSE; (*Reset TimeOut Error*)
			State   := 1003;  (*Next State*)

		ELSIF SI_Hmi_Stbd_Close.Event = INIT_CONTINUOUS THEN
			OUT_Stbd_Close := TRUE;

			TimeOut := FALSE; (*Reset TimeOut Error*)
			State   := 1004;  (*Next State*)

		END_IF

		Hyst_Old := 0;

(*	ELSIF NOT Heel_Ready AND Hyst_Old <> 1200 THEN
		IF Hyst_Cnt > CFG.Hyst_Time THEN

			OUT_Port_Open  := NOT (Port_Open AND NOT Port_Close);
			OUT_Stbd_Open  := NOT (Stbd_Open AND NOT Stbd_Close);

			Hyst_Cnt := 0.0;
			Hyst_Old := 1200;
			TimeOut  := FALSE; (*Reset TimeOut Error*)
			State    := 1200;  (*Next State*)

		ELSE
			Hyst_Cnt := Hyst_Cnt + CFG.Cycle;

		END_IF
*)

	ELSE
		(*Need to Close Port, but first be sure to open Stbd*)
		IF Heel_Value < -CFG.Hyst_HeelH AND Hyst_Old <> 1102 THEN
			IF Hyst_Cnt > CFG.Hyst_Time THEN

				OUT_Stbd_Open  := NOT (Stbd_Open AND NOT Stbd_Close);

				Hyst_Cnt := 0.0;
				Hyst_Old := 1102;
				TimeOut  := FALSE; (*Reset TimeOut Error*)
				State    := 1012;  (*Next State*)

			ELSE
				Hyst_Cnt := Hyst_Cnt + CFG.Cycle;

			END_IF

		(*Need to Close Stbd, but first be sure to open Port*)
		ELSIF Heel_Value > CFG.Hyst_HeelH AND Hyst_Old <> 1104 THEN
			IF Hyst_Cnt > CFG.Hyst_Time THEN

				OUT_Port_Open  := NOT (Port_Open AND NOT Port_Close);

				Hyst_Cnt := 0.0;
				Hyst_Old := 1104;
				TimeOut  := FALSE; (*Reset TimeOut Error*)
				State    := 1014;  (*Next State*)

			ELSE
				Hyst_Cnt := Hyst_Cnt + CFG.Cycle;

			END_IF

		ELSIF ABS(Heel_Value) < CFG.Hyst_HeelL AND Hyst_Old <> 1200 THEN
			IF Hyst_Cnt > CFG.Hyst_Time THEN

				OUT_Port_Open  := NOT (Port_Open AND NOT Port_Close);
				OUT_Stbd_Open  := NOT (Stbd_Open AND NOT Stbd_Close);
	
				Hyst_Cnt := 0.0;
				Hyst_Old := 1200;
				TimeOut  := FALSE; (*Reset TimeOut Error*)
				State    := 1200;  (*Next State*)

			ELSE
				Hyst_Cnt := Hyst_Cnt + CFG.Cycle;

			END_IF

		ELSE
			Hyst_Cnt := 0.0;

		END_IF
		(*IF ABS(Heel_Value) > CFG.Hyst_HeelH AND Hyst_Old <> 1100 THEN
			IF Hyst_Cnt > CFG.Hyst_Time THEN

				IF Heel_Value < 0 THEN

					IF Stbd_Open AND NOT Stbd_Close THEN
						OUT_Port_Close := TRUE;
					OUT_Stbd_Open  := NOT (Stbd_Open AND NOT Stbd_Close);

				ELSE
					OUT_Stbd_Close := TRUE;
					OUT_Port_Open  := NOT (Port_Open AND NOT Port_Close);

				END_IF

				Hyst_Cnt := 0.0;
				Hyst_Old := 1100;
				TimeOut  := FALSE; (*Reset TimeOut Error*)
				State    := 1100;  (*Next State*)

			ELSE
				Hyst_Cnt := Hyst_Cnt + CFG.Cycle;

			END_IF*)


	END_IF

(*Manual OUT_Port_Open*)
1001:
	IF SI_Hmi_Port_Open.Event <> NONE OR TimeOut (*OR NOT Port_Ready*) THEN
		State := 0;  (*Next State*)
	END_IF

(*Manual OUT_Port_Close*)
1002:
	IF SI_Hmi_Port_Close.Event <> NONE OR TimeOut (*OR NOT Port_Ready*) THEN
		State := 0;  (*Next State*)
	END_IF

(*Manual OUT_Stbd_Open*)
1003:
	IF SI_Hmi_Stbd_Open.Event <> NONE OR TimeOut (*OR NOT Port_Ready*) THEN
		State := 0;  (*Next State*)
	END_IF

(*Manual OUT_Stbd_Close*)
1004:
	IF SI_Hmi_Stbd_Close.Event <> NONE OR TimeOut (*OR NOT Port_Ready*) THEN
		State := 0;  (*Next State*)
	END_IF

(*Going OUT_Port_Close with Stbd Open*)
1012:
	IF NOT Heel_Ready OR Manual OR TimeOut THEN
		State := 0; (*Next State*)

	ELSIF Stbd_Open AND NOT Stbd_Close THEN
		OUT_Stbd_Open := FALSE;
		TimeCnt := 0.0;
		State   := 1102; (*Next State*)

	ELSE
		OUT_Stbd_Open := TRUE;

	END_IF

(*Going OUT_Stbd_Close with Port Open*)
1014:
	IF NOT Heel_Ready OR Manual OR TimeOut THEN
		State := 0; (*Next State*)

	ELSIF Port_Open AND NOT Port_Close THEN
		OUT_Port_Open := FALSE;
		TimeCnt := 0.0;
		State   := 1104; (*Next State*)

	ELSE
		OUT_Port_Open := TRUE;

	END_IF

(*OUT_Port_Close*)
1102:
	(*End IN*)
	IF NOT Heel_Ready OR Manual OR TimeOut THEN
		State := 0; (*Next State*)

	ELSIF Port_Close AND NOT Port_Open THEN
		State := 0; (*Next State*)

	ELSE
		OUT_Port_Close := TRUE;

	END_IF

(*OUT_Stbd_Close*)
1104:
	(*End IN*)
	IF NOT Heel_Ready OR Manual OR TimeOut THEN
		State := 0; (*Next State*)

	ELSIF Stbd_Close AND NOT Stbd_Open THEN
		State := 0; (*Next State*)

	ELSE
		OUT_Stbd_Close := TRUE;

	END_IF

(*Open Valves*)
1200:
	(*End IN*)
	IF Manual OR TimeOut THEN
		State := 0; (*Next State*)

	ELSIF (Port_Open AND NOT Port_Close) AND (Stbd_Open AND NOT Stbd_Close) THEN
		State := 0; (*Next State*)

	ELSE
		OUT_Port_Open := NOT (Port_Open AND NOT Port_Close);
		OUT_Stbd_Open := NOT (Stbd_Open AND NOT Stbd_Close);


	END_IF

END_CASE
END_FUNCTION_BLOCK

(* POU FB/FB_MAST_SETUP, ST *)
FUNCTION_BLOCK FB_MAST_SETUP
VAR_INPUT
	IN_MS  : BOOL;
	IN_1th : BOOL;
	IN_2th : BOOL;
	IN_3th : BOOL;
	IN_FH  : BOOL;

	IN_HS : BOOL;
	IN_A3 : BOOL;
	IN_F0 : BOOL;
	IN_J2 : BOOL;
	IN_J4 : BOOL;

	END_MS : BOOL;
	END_HS : BOOL;

END_VAR
VAR_IN_OUT
	FSY_P   : ST_SENSOR_BAR;
	FSY_LS  : ST_SENSOR_POS;

	BDef_P  : ST_SENSOR_BAR;
	BDef_LS : ST_SENSOR_POS;

	TDef_P  : ST_SENSOR_BAR;
	TDef_LS : ST_SENSOR_POS;

	TABLE : ST_MAST_SETUP;

END_VAR
VAR_OUTPUT
	FSY_In   : BOOL;
	FSY_Out  : BOOL;

	BDef_In  : BOOL;
	BDef_Out : BOOL;

	TDef_In  : BOOL;
	TDef_Out : BOOL;

END_VAR
VAR
	SI_MS : ARRAY[0..4] OF FB_SMART_INPUT;
	SI_HS : ARRAY[0..4] OF FB_SMART_INPUT;

	Cnt_MS : REAL;
	Cnt_HS : REAL;

	State_MS : WORD;
	State_HS : WORD;

	FSY_Tgt  : REAL;
	BDef_Tgt : REAL;
	TDef_Tgt : REAL;

END_VAR
VAR PERSISTENT
	Selected_MS AT %Q*: WORD;
	Selected_HS AT %Q*: WORD;
END_VAR
SI_MS[0](In:= IN_MS,  T_Cont:= T#1000ms, T_DClk:= T#0ms);
SI_MS[1](In:= IN_1th, T_Cont:= T#2000ms, T_DClk:= T#0ms);
SI_MS[2](In:= IN_2th, T_Cont:= T#2000ms, T_DClk:= T#0ms);
SI_MS[3](In:= IN_3th, T_Cont:= T#2000ms, T_DClk:= T#0ms);
SI_MS[4](In:= IN_FH,  T_Cont:= T#2000ms, T_DClk:= T#0ms);

SI_HS[0](In:= IN_HS, T_Cont:= T#1000ms, T_DClk:= T#0ms);
SI_HS[1](In:= IN_A3, T_Cont:= T#2000ms, T_DClk:= T#0ms);
SI_HS[2](In:= IN_F0, T_Cont:= T#2000ms, T_DClk:= T#0ms);
SI_HS[3](In:= IN_J2, T_Cont:= T#2000ms, T_DClk:= T#0ms);
SI_HS[4](In:= IN_J4, T_Cont:= T#2000ms, T_DClk:= T#0ms);

Cnt_MS := Cnt_MS + TABLE.Cycle;
Cnt_HS := Cnt_HS + TABLE.Cycle;

(*Precondition*)
IF Selected_MS < 1 OR Selected_MS > 4 THEN Selected_MS := 1; END_IF
IF Selected_HS < 1 OR Selected_HS > 6 THEN Selected_HS := 1; END_IF


(*MAIN SAIL*)
CASE State_MS OF
0:
	Cnt_MS := 0.0;

